// TIA Portal project "progetto KENNEDY_ok" (V16)

(* hardware
DEVICE "HMI_1"  KTP900 Basic PN
   slot 0: "HMI_1"  KTP900 Basic PN  6AV2 123-2JB03-0AX0  15.1.0.0
   slot 1: "HMI_RT_1"  KTP900 Basic PN  6AV2 123-2JB03-0AX0  15.1.0.0
   slot 5: "HMI_1.IE_CP_1"  PROFINET Interface  15.0.1.0
      slot 1: "Interfaccia_1 PROFINET"  PROFINET Interface
         slot 1: "Porta_1"  Port
DEVICE "S7-1200 station_1"  S7-1200 Station
   slot 0: "Telaio di montaggio_0"  S7-1200 Rack  Rack  V1.0
   slot 1: "PLC_1"  CPU 1212C DC/DC/DC  6ES7 212-1AE40-0XB0  V4.4
*)

// ===== PLC "PLC_1"  CPU 1212C DC/DC/DC =====

VAR_GLOBAL   // PLC tag table "Tabella delle variabili standard"
   "EV PISTONE 1 MISURA" AT %Q0.2 : Bool;
   "EV PINZA" AT %Q0.5 : Bool;
   "EV PISTONE 3 SU GIU" AT %Q0.4 : Bool;
   "EV PISTONE 2 MISURA" AT %Q0.3 : Bool;
   "EV AV INDIETRO RIEMPITRICE" AT %Q0.6 : Bool;
   "EV BECCUCCIO RIEMPITRICE" AT %Q0.7 : Bool;
   "EV RIEMPIMENTO FLACONE" AT %Q8.0 : Bool;
   "RISERVA 2" AT %I0.7 : Bool;
   "FC PISTONE 1 AVANTI" AT %I8.3 : Bool;
   "FC PISTONE 1 INDIETRO" AT %I8.4 : Bool;
   "FC PISTONE 2 AVANTI" AT %I8.5 : Bool;
   "FC PISTONE 2 INDIETRO" AT %I8.6 : Bool;
   "FC PISTONE 3 VERTICALE GIU" AT %I8.7 : Bool;
   "FC PISTONE 3 VERTICALE SU" AT %I9.0 : Bool;
   "FC PISTONE 4 PINZA APERTA" AT %I9.1 : Bool;
   "FC SENSORE PRESENZA PEZZO AL CARICO" AT %I9.2 : Bool;
   "FUNGO EMERGENZA" AT %I0.0 : Bool;
   "PULSANTE RESET EMERGENZA" AT %I0.1 : Bool;
   "SELETTORE MANU  AUTO" AT %I0.3 : Bool;
   "PULSANTE START CICLO" AT %I0.4 : Bool;
   "PULSANTE STOP CICLO" AT %I0.5 : Bool;
   "RISERVA 1" AT %I0.6 : Bool;
   "PULSANTE 1" AT %I8.0 : Bool;
   "PULSANTE 2" AT %I8.1 : Bool;
   "LAMPADA RESET EMERGENZA" AT %Q0.0 : Bool;
   "LAMPADA PULSANTE START VERDE" AT %Q0.1 : Bool;
   "SELETTORE 1" AT %I0.2 : Bool;
   "FC AVANTI RIEMPITRICE" AT %I9.4 : Bool;
   "RISERVA 3" AT %I8.2 : Bool;
   "FC INDIETRO RIEMPITRICE" AT %I9.5 : Bool;
   "FC GIU BECCUCCIO RIEMPITRICE" AT %I9.6 : Bool;
   "FC SU BECCUCCIO RIEMPITRICE" AT %I9.7 : Bool;
   "Clock_Byte" AT %MB0 : Byte;
   "Clock_10Hz" AT %M0.0 : Bool;
   "Clock_5Hz" AT %M0.1 : Bool;
   "Clock_2.5Hz" AT %M0.2 : Bool;
   "Clock_2Hz" AT %M0.3 : Bool;
   "Clock_1.25Hz" AT %M0.4 : Bool;
   "Clock_1Hz" AT %M0.5 : Bool;
   "Clock_0.625Hz" AT %M0.6 : Bool;
   "Clock_0.5Hz" AT %M0.7 : Bool;
   "RISERVA 4" AT %I9.3 : Bool;
END_VAR

DATA_BLOCK "0-DB-Generale"   // DB4
{ S7_Optimized_Access := 'TRUE' }
VERSION : 0.1
   VAR
      "0-COMMENTO" : Bool;   // Usata per decommentare righe di ladder
      "0-TEST" : Bool;   // Usata per simulare una uscita finta nei test
      "0-IdCommessa" : Int;   // Identificiativo della commessa (ipoteticamente) ricevuta dal pc bordo macchina
      "0-IdMacchinario" : Int;   // Int da fissare costante all'interno della macchina. Identifica univocamente il PLC, ma noi ne abbiamo uno solo
      "0-IdProdotto" : Int;   // Identificativo del prodotto (ipoteticamente) commissionato dall'ufficio
      "0-PezziTotali" : Int;   // Il numero toale di pezzi da produrre (ipoteticamente impostato da ufficio)
      "0-TimeStampAttuale" : DTL;   // Il tempo reale del plc
      "0-PezziBuoniProdotti" : Int;   // Il numero di pezzi non difettati prodotti
      "0-PezziScartiProdotti" : Int;   // Il numero di pezzi fallati prodotti
      "0-StatoMacchina" : Int;   // L'intero in sostituziona all'enum che identifica lo stato macchina: viene gestito (prelevato tramite OPC Ua e scritto in SQL Server) nel codice c#. Legenda: 0 - Verde, Stato Start; 1 - Rosso, Stato Fermo; 2 - Giallo, Stato Pronto;
      "0-MinutiDiLavoro" : Int;   // I minuti totali di lavoro del macchinario: sono dati dall'accumulo delle differenze tra TImeStampFineCiclo e TImeStampInizioCiclo alla fine di ogni ciclo
      "0-TImeStampInizioCiclo" : Int;   // TimeStamp al momento dell'inizio del ciclo di una data commessa
      "0-TimeStampFineCiclo" : Int;   // TimeStamp al momento della fine del ciclo di una data commessa
      "0-IdAttuatori" : Array[0..1] of Int;   // Id univoco per ciascun pistoni in questo PLC (idealmente potrebbe tracciare anche singole parti meccaniche come viti ecc. ecc.). E' analogo al mac address delle schede di rete nei pc per intendersi.
      "0-NumeroAttivazioniAttuatori" : Array[0..1] of Int;   // Array che contiene l'accumulatore delle attivazioni degli attuatori per ciascun attuatore. In altre parole mi immagino una matrice con una riga con l'array degli attuatori e una riga sotto con l'accumulo delle attivazioni per ogni attuatore
      "0-IdSensori" : Array[0..1] of Int;   // Analogo agli attuatori: vedi loro commenti
      "0-NumeroAttivazioniSensori" : Array[0..1] of Int;   // Analogo agli attuatori: vedi loro commenti
      "0-PezziPerMinuto" : Real;   // Usiamo l'equivalente PLC del float. Per standard contrattuali e' buona pratica usare il tipo REAL per le velocita' al minuto
      "0-Allarmi" : Array[0..1] of Bool;   // Attivazione o Meno di ogni allarme (logica simile alla matrice deglia attuatori: vedi commenti sopra)
      "1-NonEmergenza" : Bool;   // NonEmergenza = True = macchina in regolare funzione, NonEmergenza = False = macchina in emergenza e ferma
      "3-AvvioCicloAuto" : Bool;   // Il ciclo automatico si avvia
      "3-CicloAutoPronto" : Bool;   // Il ciclo automatico e' pronto per l'avvio
      "3-MacchinaInPosizioneDiPartenza" : Bool;   // Risultato logico combinatorio sui finecorsa (se sono tutti nelle opportune posizioni la macchina e' nella posizione iniziale)
      "3-GestioneManuPronta" : Bool;   // La gestione manuale dell'automazione da hmi e' pronta per essere usata
      "3-AvvioGestioneManu" : Bool;   // La gestione manuale si avvia
      "4-ResetMacchinaInPosizioneDiPartenza" : Bool;   // Resetta le posizioni dei pistoni alla fine del ciclo
      "4-Passo1" : Bool;   // Il pistone 3 si abbassa sul flacone (pre riempimento)
      "4-Passo2" : Bool;   // Il pistone Pinza si chiude sul flacone (pre riempimento)
      "4-Passo3" : Bool;   // Il pistone 3 si alza con il flacone (pre riempimento)
      "4-Passo4" : Bool;   // Il pistone 2 si estende a destra (pre riempimento)
      "4-Passo5" : Bool;   // Il pistone 1 si estende a destra (pre riempimento)
      "4-Passo6" : Bool;   // Il pistone 3 si abbassa con il flacone (pre riempimento)
      "4-Passo7" : Bool;   // Il pistone pinza si apre con il flacone (pre riempimento)
      "4-Passo8" : Bool;   // Il pistone 3 si alza senza flacone in attesa del riempimento (pre riempimento)
      "4-Passo9" : Bool;   // Il pistone riempitore 1 si estende a sinistra
      "4-Passo10" : Bool;   // Il pistone riempitore 2 abbassa il beccuccio
      "4-Passo11" : Bool;   // Il pistone riempitore 2 alza il beccuccio
      "4-Passo12" : Bool;   // Il pistone riempitore 1 rientra a destra
      "4-Passo13" : Bool;   // Il pistone 3 scende sopra al flacone (post riempimento)
      "4-Passo14" : Bool;   // Il pistone Pinza si chiude sul flacone (post riempimento)
      "4-Passo15" : Bool;   // Il pistone 3 si alza con il flacone (post riempimento)
      "4-Passo16" : Bool;   // Il pistone 2 si ritrae con il flacone (post riempimento)
      "4-Passo17" : Bool;   // Il pistone 3 si abbassa sulla zona di scarico
      "4-Passo18" : Bool;   // Il pistone Pinza si apre
      "4-Passo19" : Bool;   // Il pistone 3 si alza dalla zona di scarico
      "4-Passo20" : Bool;   // Il pistone 1 si ritrae nella posizione di partenza: il ciclo è finito
      "5-HMI => Only current time" : Time_Of_Day;   // Ora corrente (time) estrapolata dal dato totale (Time of Day)
      "5-HMI => Only current date" : Date;   // Data corrente (date) estrapolata dal dato totale (Time of Day)
      "5-HMI => Current time of day" : DTL;   // Current Time of Day include tutti i dati temporali all'acquisizione, è una sorta di TimeStamp, tipo dato DTL
      "5-HMI => Timer ultima eccezione" : Bool;   // Variabile che gestisce l'obbligo di esecuzione del login: compare un messaggio temporizzato a 5s ogni volta che si cliccano elementi cliccabili nell'HMI senza effettuare il login
      "5-ErroriDiConversione" : Int;   // Qui vengono ritornati gli interi che indicano eventuali errori nella conversione ed estrazione di data o ora dalla DTL che contiene tutto il timestamp. Se la conversione avviene con successo il valore di questa variabile è 0000
      "5-VisibilitaComandiManuali" : Bool;   // Gestisce la visibilita' dell'automazione per la schermata manuale dell'hmi. In base allo stato della variabile si vede il manipolatore o la riempitrice.
      "6-Pistone-1-Manuale" : Bool;   // Variabile d'appoggio a sostituire l'uscita diretta nel blocco ciclo manuale
      "6-Pistone-2-Manuale" : Bool;   // Variabile d'appoggio a sostituire l'uscita diretta nel blocco ciclo manuale
      "6-Pistone-3-Manuale" : Bool;   // Variabile d'appoggio a sostituire l'uscita diretta nel blocco ciclo manuale
      "6-Pistone-4-(Pinza)-Manuale" : Bool;   // Variabile d'appoggio a sostituire l'uscita diretta nel blocco ciclo manuale
      "6-Pistone-5-(Riempitrice)-Manuale" : Bool;   // Variabile d'appoggio a sostituire l'uscita diretta nel blocco ciclo manuale
      "6-Beccuccio-(Riempitrice)-Manuale" : Bool;   // Variabile d'appoggio a sostituire l'uscita diretta nel blocco ciclo manuale
      "6-Riempimento-(Riempitrice)-Manuale" : Bool;   // Variabile d'appoggio a sostituire l'uscita diretta nel blocco ciclo manuale
      "6-PulsanteAvantiPistone1" : Bool;   // Variabile d'appoggio che identifica il relativo tasto dell'HMI nel blocco uscite
      "6-PulsanteIndietroPistone1" : Bool;   // Variabile d'appoggio che identifica il relativo tasto dell'HMI nel blocco uscite
      "6-PulsanteAvantiPistone2" : Bool;   // Variabile d'appoggio che identifica il relativo tasto dell'HMI nel blocco uscite
      "6-PulsanteIndietroPistone2" : Bool;   // Variabile d'appoggio che identifica il relativo tasto dell'HMI nel blocco uscite
      "6-PulsanteGiuPistone3" : Bool;   // Variabile d'appoggio che identifica il relativo tasto dell'HMI nel blocco uscite
      "6-PulsanteSuPistone3" : Bool;   // Variabile d'appoggio che identifica il relativo tasto dell'HMI nel blocco uscite
      "6-PulsanteChiudiPinza" : Bool;   // Variabile d'appoggio che identifica il relativo tasto dell'HMI nel blocco uscite
      "6-PulsanteApriPinza" : Bool;   // Variabile d'appoggio che identifica il relativo tasto dell'HMI nel blocco uscite
      "6-PulsanteAvantiPistone5Riempitrice" : Bool;   // Variabile d'appoggio che identifica il relativo tasto dell'HMI nel blocco uscite
      "6-PulsanteIndietroPistone5Riempitrice" : Bool;   // Variabile d'appoggio che identifica il relativo tasto dell'HMI nel blocco uscite
      "6-PulsanteGiuPistone6Beccuccio" : Bool;   // Variabile d'appoggio che identifica il relativo tasto dell'HMI nel blocco uscite
      "6-PulsanteSuPistone6Beccuccio" : Bool;   // Variabile d'appoggio che identifica il relativo tasto dell'HMI nel blocco uscite
      "6-PulsanteRiempimento" : Bool;
   END_VAR
BEGIN
END_DATA_BLOCK

// folder: RISERVATO_NON_MODIFICARE

DATA_BLOCK "Blocco_dati_1"   // DB1
{ S7_Optimized_Access := 'TRUE' }
VERSION : 0.1
   VAR
      "pistone 1  X" : Int;
      "pistone 1  Y" : Int;
      "pistone 2  X" : Int;
      "pistone 2 Y" : Int;
      "stelo pistone 2 x" : Int;
      "stelo pistone 2 y" : Int;
      "pistone 3  X" : Int;
      "pistone 3 Y" : Int;
      "stelo pistone 3 x" : Int;
      "stelo pistone 3 y" : Int;
      "corpo pinza x" : Int;
      "corpo pinza y" : Int;
      "dita aperte x" : Int;
      "dita aperte y" : Int;
      "dita chiuse x" : Int;
      "dita chiuse y" : Int;
      "pistone riempitore av ind x" : Int;
      "pistone riempitore av ind y" : Int;
      "riempitore av ind x" : Int;
      "riempitore su giu y" : Int;
      "flacone x" : Int;
      "flacone y" : Int;
      "riempimento flacone" : Int;
      "pinza aperta" : Int;
      "pinza chiusa" : Int;
      "fungo emergenza" : Bool;
      "reset emergenza" : Bool;
      "lampada emergenza" : Bool;
      "pulsante start ciclo" : Bool;
      "lampada pulsante start ciclo" : Bool;
      "selettore 1 leva corta" : Bool;
      "selettore auto manu" : Bool;
      "pulsante 1" : Bool;
      "pulsante 2" : Bool;
      "pulsante stop ciclo" : Bool;
      MANUALI : Byte;
      "FLACONE PIENO" : Bool;
      "FLACONE PRESO" : Bool;
      "FLACONE IN RIEMPIMENTO" : Bool;
      "SENSORE SU" : Byte;
      "SENSORE GIU" : Byte;
      "SENSORE PINZA APERTA" : Byte;
      "SENSORE INDIETRO PISTONE_1" : Byte;
      "SENSORE AVANTI PISTONE_1" : Byte;
      "SENSORE INDIETRO PISTONE_2" : Byte;
      "SENSORE AVANTI PISTONE_2" : Byte;
      "SENSORE INDIETRO PISTONE_3" : Byte;
      "SENSORE AVANTI PISTONE_3" : Byte;
      "SENSORE INDIETRO RIEMPITRICE" : Byte;
      "SENSORE AVANTI RIEMPITRICE" : Byte;
      "SENSORE SU RIEMPITRICE" : Byte;
      "SENSORE GIU RIEMPITRICE" : Byte;
      "SENSORE PRESENZA FLACONE" : Bool;
      "RISPOSTA TELECAMERA DI ISPEZIONE" : Byte;
      "APPOGGIO PARTENZA" : Bool;
      "SELETTORE SIMULAZIONE PRESENZA PEZZO AL CARICO" : Bool;
      "VISUALIZZA IL FLACONE" : Bool;
   END_VAR
BEGIN
END_DATA_BLOCK

// folder: System blocks/Program resources

DATA_BLOCK "IEC_Timer_0_DB"   // DB2
{ S7_Optimized_Access := 'TRUE' }
AUTHOR : Simatic
FAMILY : IEC
NAME : IEC_TMR
VERSION : 1.0
// stored: InstanceOfName IEC_TIMER
"IEC_TIMER"
BEGIN
END_DATA_BLOCK

DATA_BLOCK "azzerooo"   // DB3
{ S7_Optimized_Access := 'TRUE' }
AUTHOR : Simatic
FAMILY : IEC
NAME : IEC_TMR
VERSION : 1.0
// stored: InstanceOfName IEC_TIMER
"IEC_TIMER"
BEGIN
END_DATA_BLOCK

DATA_BLOCK "IEC_Timer_0_DB_3"   // DB5
{ S7_Optimized_Access := 'TRUE' }
AUTHOR : Simatic
FAMILY : IEC
NAME : IEC_TMR
VERSION : 1.0
// stored: InstanceOfName IEC_TIMER
"IEC_TIMER"
BEGIN
END_DATA_BLOCK

DATA_BLOCK "IEC_Timer_0_DB_4"   // DB6
{ S7_Optimized_Access := 'TRUE' }
AUTHOR : Simatic
FAMILY : IEC
NAME : IEC_TMR
VERSION : 1.0
// stored: InstanceOfName IEC_TIMER
"IEC_TIMER"
BEGIN
END_DATA_BLOCK

DATA_BLOCK "IEC_Timer_0_DB_5"   // DB7
{ S7_Optimized_Access := 'TRUE' }
AUTHOR : Simatic
FAMILY : IEC
NAME : IEC_TMR
VERSION : 1.0
// stored: InstanceOfName IEC_TIMER
"IEC_TIMER"
BEGIN
END_DATA_BLOCK

DATA_BLOCK "IEC_Timer_0_DB_6"   // DB8
{ S7_Optimized_Access := 'TRUE' }
AUTHOR : Simatic
FAMILY : IEC
NAME : IEC_TMR
VERSION : 1.0
// stored: InstanceOfName IEC_TIMER
"IEC_TIMER"
BEGIN
END_DATA_BLOCK

DATA_BLOCK "IEC_Timer_0_DB_7"   // DB9
{ S7_Optimized_Access := 'TRUE' }
AUTHOR : Simatic
FAMILY : IEC
NAME : IEC_TMR
VERSION : 1.0
// stored: InstanceOfName IEC_TIMER
"IEC_TIMER"
BEGIN
END_DATA_BLOCK

DATA_BLOCK "IEC_Timer_0_DB_8"   // DB10
{ S7_Optimized_Access := 'TRUE' }
AUTHOR : Simatic
FAMILY : IEC
NAME : IEC_TMR
VERSION : 1.0
// stored: InstanceOfName IEC_TIMER
"IEC_TIMER"
BEGIN
END_DATA_BLOCK

DATA_BLOCK "IEC_Timer_0_DB_9"   // DB11
{ S7_Optimized_Access := 'TRUE' }
AUTHOR : Simatic
FAMILY : IEC
NAME : IEC_TMR
VERSION : 1.0
// stored: InstanceOfName IEC_TIMER
"IEC_TIMER"
BEGIN
END_DATA_BLOCK

DATA_BLOCK "IEC_Timer_0_DB_10"   // DB12
{ S7_Optimized_Access := 'TRUE' }
AUTHOR : Simatic
FAMILY : IEC
NAME : IEC_TMR
VERSION : 1.0
// stored: InstanceOfName IEC_TIMER
"IEC_TIMER"
BEGIN
END_DATA_BLOCK

DATA_BLOCK "IEC_Timer_0_DB_11"   // DB13
{ S7_Optimized_Access := 'TRUE' }
AUTHOR : Simatic
FAMILY : IEC
NAME : IEC_TMR
VERSION : 1.0
// stored: InstanceOfName IEC_TIMER
"IEC_TIMER"
BEGIN
END_DATA_BLOCK

DATA_BLOCK "IEC_Timer_0_DB_12"   // DB14
{ S7_Optimized_Access := 'TRUE' }
AUTHOR : Simatic
FAMILY : IEC
NAME : IEC_TMR
VERSION : 1.0
// stored: InstanceOfName IEC_TIMER
"IEC_TIMER"
BEGIN
END_DATA_BLOCK

DATA_BLOCK "IEC_Timer_0_DB_13"   // DB15
{ S7_Optimized_Access := 'TRUE' }
AUTHOR : Simatic
FAMILY : IEC
NAME : IEC_TMR
VERSION : 1.0
// stored: InstanceOfName IEC_TIMER
"IEC_TIMER"
BEGIN
END_DATA_BLOCK

DATA_BLOCK "IEC_Timer_0_DB_1"   // DB16
{ S7_Optimized_Access := 'TRUE' }
AUTHOR : Simatic
FAMILY : IEC
NAME : IEC_TMR
VERSION : 1.0
// stored: InstanceOfName IEC_TIMER
"IEC_TIMER"
BEGIN
END_DATA_BLOCK

DATA_BLOCK "IEC_Timer_0_DB_2"   // DB17
{ S7_Optimized_Access := 'TRUE' }
AUTHOR : Simatic
FAMILY : IEC
NAME : IEC_TMR
VERSION : 1.0
// stored: InstanceOfName IEC_TIMER
"IEC_TIMER"
BEGIN
END_DATA_BLOCK

DATA_BLOCK "IEC_Timer_0_DB_14"   // DB18
{ S7_Optimized_Access := 'TRUE' }
AUTHOR : Simatic
FAMILY : IEC
NAME : IEC_TMR
VERSION : 1.0
// stored: InstanceOfName IEC_TIMER
"IEC_TIMER"
BEGIN
END_DATA_BLOCK

DATA_BLOCK "IEC_Timer_0_DB_15"   // DB19
{ S7_Optimized_Access := 'TRUE' }
AUTHOR : Simatic
FAMILY : IEC
NAME : IEC_TMR
VERSION : 1.0
// stored: InstanceOfName IEC_TIMER
"IEC_TIMER"
BEGIN
END_DATA_BLOCK

DATA_BLOCK "IEC_Timer_0_DB_16"   // DB20
{ S7_Optimized_Access := 'TRUE' }
AUTHOR : Simatic
FAMILY : IEC
NAME : IEC_TMR
VERSION : 1.0
// stored: InstanceOfName IEC_TIMER
"IEC_TIMER"
BEGIN
END_DATA_BLOCK

DATA_BLOCK "IEC_Timer_0_DB_17"   // DB21
{ S7_Optimized_Access := 'TRUE' }
AUTHOR : Simatic
FAMILY : IEC
NAME : IEC_TMR
VERSION : 1.0
// stored: InstanceOfName IEC_TIMER
"IEC_TIMER"
BEGIN
END_DATA_BLOCK

DATA_BLOCK "IEC_Timer_0_DB_18"   // DB22
{ S7_Optimized_Access := 'TRUE' }
AUTHOR : Simatic
FAMILY : IEC
NAME : IEC_TMR
VERSION : 1.0
// stored: InstanceOfName IEC_TIMER
"IEC_TIMER"
BEGIN
END_DATA_BLOCK

DATA_BLOCK "IEC_Timer_0_DB_19"   // DB23
{ S7_Optimized_Access := 'TRUE' }
AUTHOR : Simatic
FAMILY : IEC
NAME : IEC_TMR
VERSION : 1.0
// stored: InstanceOfName IEC_TIMER
"IEC_TIMER"
BEGIN
END_DATA_BLOCK

DATA_BLOCK "IEC_Timer_0_DB_20"   // DB24
{ S7_Optimized_Access := 'TRUE' }
AUTHOR : Simatic
FAMILY : IEC
NAME : IEC_TMR
VERSION : 1.0
// stored: InstanceOfName IEC_TIMER
"IEC_TIMER"
BEGIN
END_DATA_BLOCK

DATA_BLOCK "IEC_Timer_0_DB_21"   // DB25
{ S7_Optimized_Access := 'TRUE' }
AUTHOR : Simatic
FAMILY : IEC
NAME : IEC_TMR
VERSION : 1.0
// stored: InstanceOfName IEC_TIMER
"IEC_TIMER"
BEGIN
END_DATA_BLOCK

DATA_BLOCK "IEC_Timer_0_DB_22"   // DB26
{ S7_Optimized_Access := 'TRUE' }
AUTHOR : Simatic
FAMILY : IEC
NAME : IEC_TMR
VERSION : 1.0
// stored: InstanceOfName IEC_TIMER
"IEC_TIMER"
BEGIN
END_DATA_BLOCK

DATA_BLOCK "IEC_Timer_0_DB_23"   // DB27
{ S7_Optimized_Access := 'TRUE' }
AUTHOR : Simatic
FAMILY : IEC
NAME : IEC_TMR
VERSION : 1.0
// stored: InstanceOfName IEC_TIMER
"IEC_TIMER"
BEGIN
END_DATA_BLOCK

DATA_BLOCK "IEC_Timer_0_DB_24"   // DB28
{ S7_Optimized_Access := 'TRUE' }
AUTHOR : Simatic
FAMILY : IEC
NAME : IEC_TMR
VERSION : 1.0
// stored: InstanceOfName IEC_TIMER
"IEC_TIMER"
BEGIN
END_DATA_BLOCK

DATA_BLOCK "IEC_Timer_0_DB_25"   // DB29
{ S7_Optimized_Access := 'TRUE' }
AUTHOR : Simatic
FAMILY : IEC
NAME : IEC_TMR
VERSION : 1.0
// stored: InstanceOfName IEC_TIMER
"IEC_TIMER"
BEGIN
END_DATA_BLOCK

DATA_BLOCK "IEC_Timer_0_DB_26"   // DB30
{ S7_Optimized_Access := 'TRUE' }
AUTHOR : Simatic
FAMILY : IEC
NAME : IEC_TMR
VERSION : 1.0
// stored: InstanceOfName IEC_TIMER
"IEC_TIMER"
BEGIN
END_DATA_BLOCK

DATA_BLOCK "IEC_Timer_0_DB_27"   // DB31
{ S7_Optimized_Access := 'TRUE' }
AUTHOR : Simatic
FAMILY : IEC
NAME : IEC_TMR
VERSION : 1.0
// stored: InstanceOfName IEC_TIMER
"IEC_TIMER"
BEGIN
END_DATA_BLOCK

DATA_BLOCK "IEC_Timer_0_DB_28"   // DB32
{ S7_Optimized_Access := 'TRUE' }
AUTHOR : Simatic
FAMILY : IEC
NAME : IEC_TMR
VERSION : 1.0
// stored: InstanceOfName IEC_TIMER
"IEC_TIMER"
BEGIN
END_DATA_BLOCK

DATA_BLOCK "IEC_Timer_0_DB_29"   // DB33
{ S7_Optimized_Access := 'TRUE' }
AUTHOR : Simatic
FAMILY : IEC
NAME : IEC_TMR
VERSION : 1.0
// stored: InstanceOfName IEC_TIMER
"IEC_TIMER"
BEGIN
END_DATA_BLOCK

DATA_BLOCK "IEC_Timer_0_DB_30"   // DB34
{ S7_Optimized_Access := 'TRUE' }
AUTHOR : Simatic
FAMILY : IEC
NAME : IEC_TMR
VERSION : 1.0
// stored: InstanceOfName IEC_TIMER
"IEC_TIMER"
BEGIN
END_DATA_BLOCK

DATA_BLOCK "IEC_Timer_0_DB_31"   // DB35
{ S7_Optimized_Access := 'TRUE' }
AUTHOR : Simatic
FAMILY : IEC
NAME : IEC_TMR
VERSION : 1.0
// stored: InstanceOfName IEC_TIMER
"IEC_TIMER"
BEGIN
END_DATA_BLOCK

DATA_BLOCK "IEC_Timer_0_DB_32"   // DB36
{ S7_Optimized_Access := 'TRUE' }
AUTHOR : Simatic
FAMILY : IEC
NAME : IEC_TMR
VERSION : 1.0
// stored: InstanceOfName IEC_TIMER
"IEC_TIMER"
BEGIN
END_DATA_BLOCK

DATA_BLOCK "IEC_Timer_0_DB_33"   // DB37
{ S7_Optimized_Access := 'TRUE' }
AUTHOR : Simatic
FAMILY : IEC
NAME : IEC_TMR
VERSION : 1.0
// stored: InstanceOfName IEC_TIMER
"IEC_TIMER"
BEGIN
END_DATA_BLOCK

DATA_BLOCK "IEC_Timer_0_DB_34"   // DB38
{ S7_Optimized_Access := 'TRUE' }
AUTHOR : Simatic
FAMILY : IEC
NAME : IEC_TMR
VERSION : 1.0
// stored: InstanceOfName IEC_TIMER
"IEC_TIMER"
BEGIN
END_DATA_BLOCK

// folder: (top level)

FUNCTION "1-Allarmi" : Void   // FC2, LAD
{ S7_Optimized_Access := 'TRUE' }
VERSION : 0.1
BEGIN

REGION Network 1: NonEmergenza = True = macchina in regolare funzione, NonEmergenza = False = macchina in emergenza e ferma
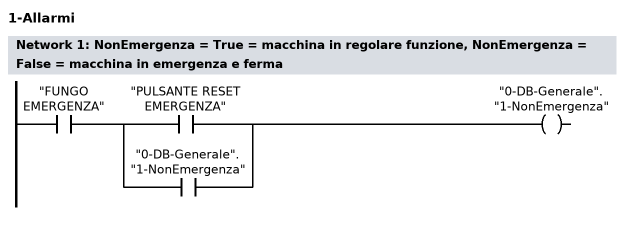
   RUNG wire#powerrail
      Contact( "FUNGO EMERGENZA" )
      wire#w1
      Contact( "PULSANTE RESET EMERGENZA" )
      wire#w2
      Coil( "0-DB-Generale"."1-NonEmergenza" )
   END_RUNG
   RUNG wire#w1
      Contact( "0-DB-Generale"."1-NonEmergenza" )
   END_RUNG wire#w2
   // the same network as SCL:
   "0-DB-Generale"."1-NonEmergenza" := "FUNGO EMERGENZA" AND ("PULSANTE RESET EMERGENZA" OR "0-DB-Generale"."1-NonEmergenza");
END_REGION
END_FUNCTION

FUNCTION "2-Uscite" : Void   // FC3, LAD
{ S7_Optimized_Access := 'TRUE' }
VERSION : 0.1
BEGIN

REGION Network 1: USCITA %Q0.0 - LAMPADA DI EMERGENZA
   // Descr: 
   // Who: Gestione prima uscita cablata.
   // What: Se la macchina non è in emergenza la lampada non si accende e viceversa.
   // How: Verifica mediante test ladder True If Off (--|/|--, NC) sulla variabile booleana (bit) associata allo stato di emergenza. Se il fungo viene usato lo stato di NonEmergenza passa da 1 a 0, da true a false quindi qui il True If Off lascia passare il segnale attivando la lampada reset di emergenza.
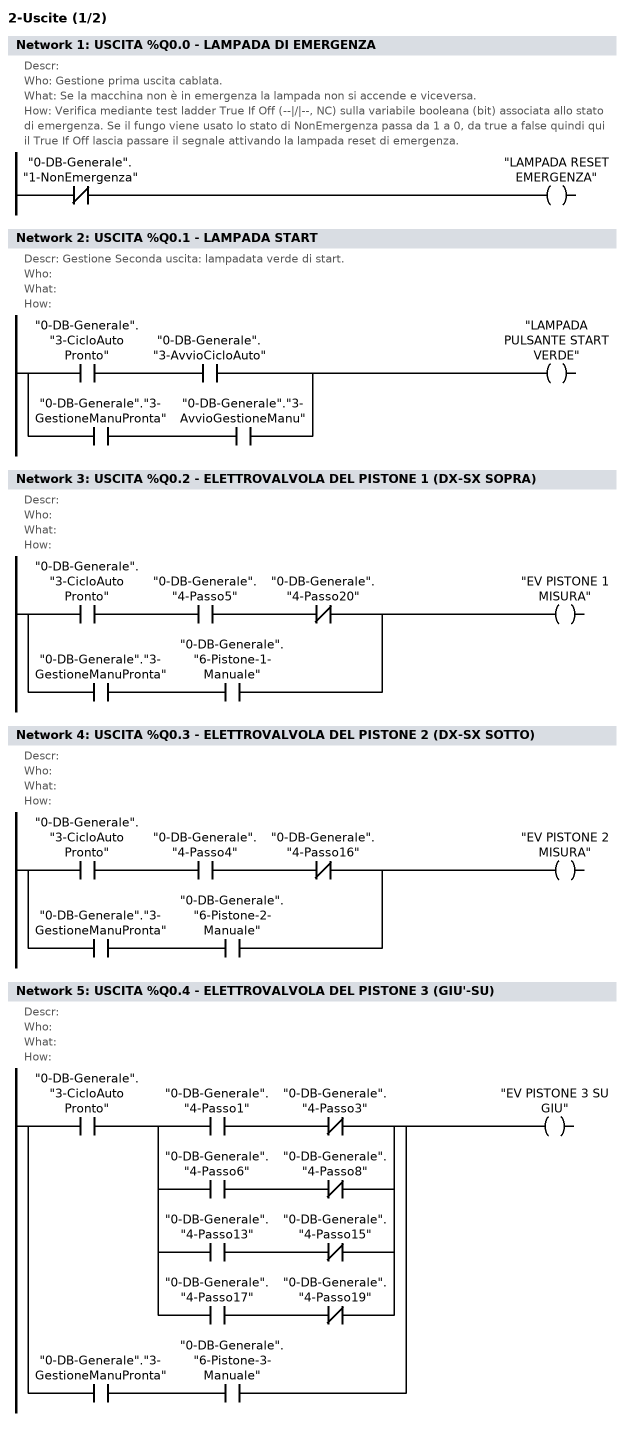
   RUNG wire#powerrail
      I_Contact( "0-DB-Generale"."1-NonEmergenza" )
      Coil( "LAMPADA RESET EMERGENZA" )
   END_RUNG
   // the same network as SCL:
   "LAMPADA RESET EMERGENZA" := NOT "0-DB-Generale"."1-NonEmergenza";
END_REGION

REGION Network 2: USCITA %Q0.1 - LAMPADA START
   // Descr: Gestione Seconda uscita: lampadata verde di start.
   // Who: 
   // What: 
   // How:
   RUNG wire#powerrail
      Contact( "0-DB-Generale"."3-CicloAutoPronto" )
      Contact( "0-DB-Generale"."3-AvvioCicloAuto" )
      wire#w1
      Coil( "LAMPADA PULSANTE START VERDE" )
   END_RUNG
   RUNG wire#powerrail
      Contact( "0-DB-Generale"."3-GestioneManuPronta" )
      Contact( "0-DB-Generale"."3-AvvioGestioneManu" )
   END_RUNG wire#w1
   // the same network as SCL:
   "LAMPADA PULSANTE START VERDE" := ("0-DB-Generale"."3-CicloAutoPronto" AND "0-DB-Generale"."3-AvvioCicloAuto") OR ("0-DB-Generale"."3-GestioneManuPronta" AND "0-DB-Generale"."3-AvvioGestioneManu");
END_REGION

REGION Network 3: USCITA %Q0.2 - ELETTROVALVOLA DEL PISTONE 1 (DX-SX SOPRA)
   // Descr: 
   // Who: 
   // What: 
   // How:
   RUNG wire#powerrail
      Contact( "0-DB-Generale"."3-CicloAutoPronto" )
      Contact( "0-DB-Generale"."4-Passo5" )
      I_Contact( "0-DB-Generale"."4-Passo20" )
      wire#w1
      Coil( "EV PISTONE 1 MISURA" )
   END_RUNG
   RUNG wire#powerrail
      Contact( "0-DB-Generale"."3-GestioneManuPronta" )
      Contact( "0-DB-Generale"."6-Pistone-1-Manuale" )
   END_RUNG wire#w1
   // the same network as SCL:
   "EV PISTONE 1 MISURA" := ("0-DB-Generale"."3-CicloAutoPronto" AND "0-DB-Generale"."4-Passo5" AND NOT "0-DB-Generale"."4-Passo20") OR ("0-DB-Generale"."3-GestioneManuPronta" AND "0-DB-Generale"."6-Pistone-1-Manuale");
END_REGION

REGION Network 4: USCITA %Q0.3 - ELETTROVALVOLA DEL PISTONE 2 (DX-SX SOTTO)
   // Descr: 
   // Who: 
   // What: 
   // How:
   RUNG wire#powerrail
      Contact( "0-DB-Generale"."3-CicloAutoPronto" )
      Contact( "0-DB-Generale"."4-Passo4" )
      I_Contact( "0-DB-Generale"."4-Passo16" )
      wire#w1
      Coil( "EV PISTONE 2 MISURA" )
   END_RUNG
   RUNG wire#powerrail
      Contact( "0-DB-Generale"."3-GestioneManuPronta" )
      Contact( "0-DB-Generale"."6-Pistone-2-Manuale" )
   END_RUNG wire#w1
   // the same network as SCL:
   "EV PISTONE 2 MISURA" := ("0-DB-Generale"."3-CicloAutoPronto" AND "0-DB-Generale"."4-Passo4" AND NOT "0-DB-Generale"."4-Passo16") OR ("0-DB-Generale"."3-GestioneManuPronta" AND "0-DB-Generale"."6-Pistone-2-Manuale");
END_REGION

REGION Network 5: USCITA %Q0.4 - ELETTROVALVOLA DEL PISTONE 3 (GIU'-SU)
   // Descr: 
   // Who: 
   // What: 
   // How:
   RUNG wire#powerrail
      Contact( "0-DB-Generale"."3-CicloAutoPronto" )
      wire#w1
      Contact( "0-DB-Generale"."4-Passo1" )
      I_Contact( "0-DB-Generale"."4-Passo3" )
      wire#w2
      Coil( "EV PISTONE 3 SU GIU" )
   END_RUNG
   RUNG wire#w1
      Contact( "0-DB-Generale"."4-Passo6" )
      I_Contact( "0-DB-Generale"."4-Passo8" )
   END_RUNG wire#w2
   RUNG wire#w1
      Contact( "0-DB-Generale"."4-Passo13" )
      I_Contact( "0-DB-Generale"."4-Passo15" )
   END_RUNG wire#w2
   RUNG wire#w1
      Contact( "0-DB-Generale"."4-Passo17" )
      I_Contact( "0-DB-Generale"."4-Passo19" )
   END_RUNG wire#w2
   RUNG wire#powerrail
      Contact( "0-DB-Generale"."3-GestioneManuPronta" )
      Contact( "0-DB-Generale"."6-Pistone-3-Manuale" )
   END_RUNG wire#w2
   // the same network as SCL:
   "EV PISTONE 3 SU GIU" := ("0-DB-Generale"."3-CicloAutoPronto" AND (("0-DB-Generale"."4-Passo1" AND NOT "0-DB-Generale"."4-Passo3") OR ("0-DB-Generale"."4-Passo6" AND NOT "0-DB-Generale"."4-Passo8") OR ("0-DB-Generale"."4-Passo13" AND NOT "0-DB-Generale"."4-Passo15") OR ("0-DB-Generale"."4-Passo17" AND NOT "0-DB-Generale"."4-Passo19"))) OR ("0-DB-Generale"."3-GestioneManuPronta" AND "0-DB-Generale"."6-Pistone-3-Manuale");
END_REGION

REGION Network 6: USCITA %Q0.5 - ELETTROVALVOLA DELLA PINZA (APRI-CHIUDI)
   // Descr: 
   // Who: 
   // What: 
   // How:
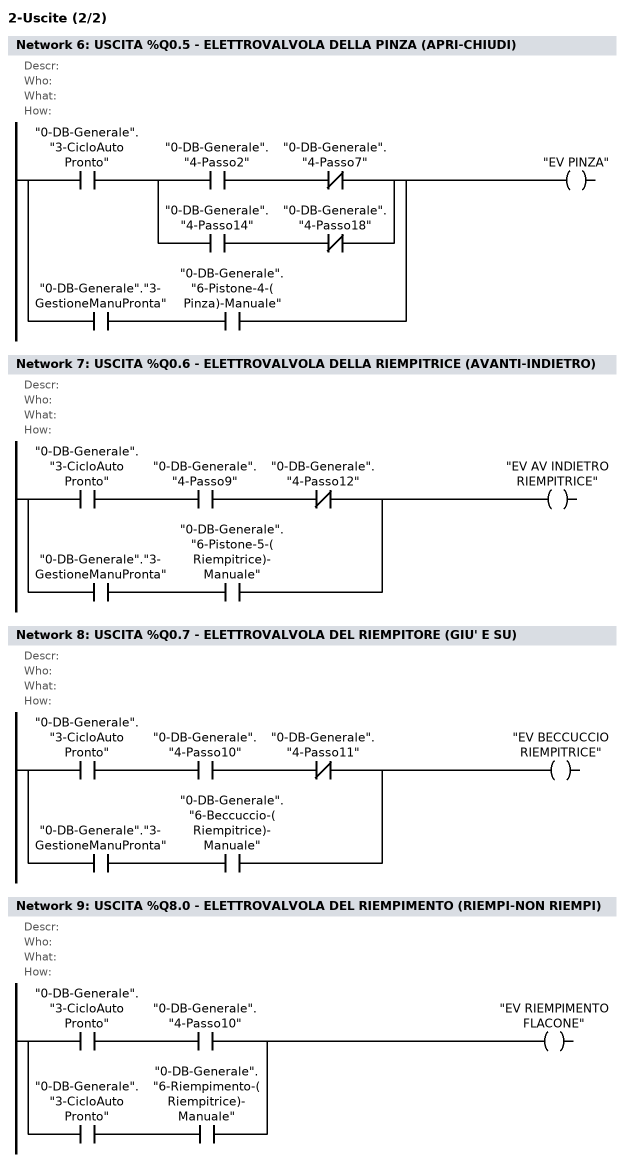
   RUNG wire#powerrail
      Contact( "0-DB-Generale"."3-CicloAutoPronto" )
      wire#w1
      Contact( "0-DB-Generale"."4-Passo2" )
      I_Contact( "0-DB-Generale"."4-Passo7" )
      wire#w2
      Coil( "EV PINZA" )
   END_RUNG
   RUNG wire#w1
      Contact( "0-DB-Generale"."4-Passo14" )
      I_Contact( "0-DB-Generale"."4-Passo18" )
   END_RUNG wire#w2
   RUNG wire#powerrail
      Contact( "0-DB-Generale"."3-GestioneManuPronta" )
      Contact( "0-DB-Generale"."6-Pistone-4-(Pinza)-Manuale" )
   END_RUNG wire#w2
   // the same network as SCL:
   "EV PINZA" := ("0-DB-Generale"."3-CicloAutoPronto" AND (("0-DB-Generale"."4-Passo2" AND NOT "0-DB-Generale"."4-Passo7") OR ("0-DB-Generale"."4-Passo14" AND NOT "0-DB-Generale"."4-Passo18"))) OR ("0-DB-Generale"."3-GestioneManuPronta" AND "0-DB-Generale"."6-Pistone-4-(Pinza)-Manuale");
END_REGION

REGION Network 7: USCITA %Q0.6 - ELETTROVALVOLA DELLA RIEMPITRICE (AVANTI-INDIETRO)
   // Descr: 
   // Who: 
   // What: 
   // How:
   RUNG wire#powerrail
      Contact( "0-DB-Generale"."3-CicloAutoPronto" )
      Contact( "0-DB-Generale"."4-Passo9" )
      I_Contact( "0-DB-Generale"."4-Passo12" )
      wire#w1
      Coil( "EV AV INDIETRO RIEMPITRICE" )
   END_RUNG
   RUNG wire#powerrail
      Contact( "0-DB-Generale"."3-GestioneManuPronta" )
      Contact( "0-DB-Generale"."6-Pistone-5-(Riempitrice)-Manuale" )
   END_RUNG wire#w1
   // the same network as SCL:
   "EV AV INDIETRO RIEMPITRICE" := ("0-DB-Generale"."3-CicloAutoPronto" AND "0-DB-Generale"."4-Passo9" AND NOT "0-DB-Generale"."4-Passo12") OR ("0-DB-Generale"."3-GestioneManuPronta" AND "0-DB-Generale"."6-Pistone-5-(Riempitrice)-Manuale");
END_REGION

REGION Network 8: USCITA %Q0.7 - ELETTROVALVOLA DEL RIEMPITORE (GIU' E SU)
   // Descr: 
   // Who: 
   // What: 
   // How:
   RUNG wire#powerrail
      Contact( "0-DB-Generale"."3-CicloAutoPronto" )
      Contact( "0-DB-Generale"."4-Passo10" )
      I_Contact( "0-DB-Generale"."4-Passo11" )
      wire#w1
      Coil( "EV BECCUCCIO RIEMPITRICE" )
   END_RUNG
   RUNG wire#powerrail
      Contact( "0-DB-Generale"."3-GestioneManuPronta" )
      Contact( "0-DB-Generale"."6-Beccuccio-(Riempitrice)-Manuale" )
   END_RUNG wire#w1
   // the same network as SCL:
   "EV BECCUCCIO RIEMPITRICE" := ("0-DB-Generale"."3-CicloAutoPronto" AND "0-DB-Generale"."4-Passo10" AND NOT "0-DB-Generale"."4-Passo11") OR ("0-DB-Generale"."3-GestioneManuPronta" AND "0-DB-Generale"."6-Beccuccio-(Riempitrice)-Manuale");
END_REGION

REGION Network 9: USCITA %Q8.0 - ELETTROVALVOLA DEL RIEMPIMENTO (RIEMPI-NON RIEMPI)
   // Descr: 
   // Who: 
   // What: 
   // How:
   RUNG wire#powerrail
      Contact( "0-DB-Generale"."3-CicloAutoPronto" )
      Contact( "0-DB-Generale"."4-Passo10" )
      wire#w1
      Coil( "EV RIEMPIMENTO FLACONE" )
   END_RUNG
   RUNG wire#powerrail
      Contact( "0-DB-Generale"."3-CicloAutoPronto" )
      Contact( "0-DB-Generale"."6-Riempimento-(Riempitrice)-Manuale" )
   END_RUNG wire#w1
   // the same network as SCL:
   "EV RIEMPIMENTO FLACONE" := ("0-DB-Generale"."3-CicloAutoPronto" AND "0-DB-Generale"."4-Passo10") OR ("0-DB-Generale"."3-CicloAutoPronto" AND "0-DB-Generale"."6-Riempimento-(Riempitrice)-Manuale");
END_REGION
END_FUNCTION

FUNCTION "3-AvvioAutoManu" : Void   // FC4, LAD
TITLE = NETWORK 1-3: AVVIO CICLO AUTOMATICO; NETWORK 4-5: AVVIO GESTIONE MANUALE
{ S7_Optimized_Access := 'TRUE' }
VERSION : 0.1
BEGIN

REGION Network 1: CONTROLLO SE L'AUTOMAZIONE E' PRONTA AD AVVIARE IL CICLO AUTOMATICO
   // Se la macchina non è in emergenza E il selettore Manu/Auto è in Automatico allora la macchina è pronta per avviare il ciclo automatico
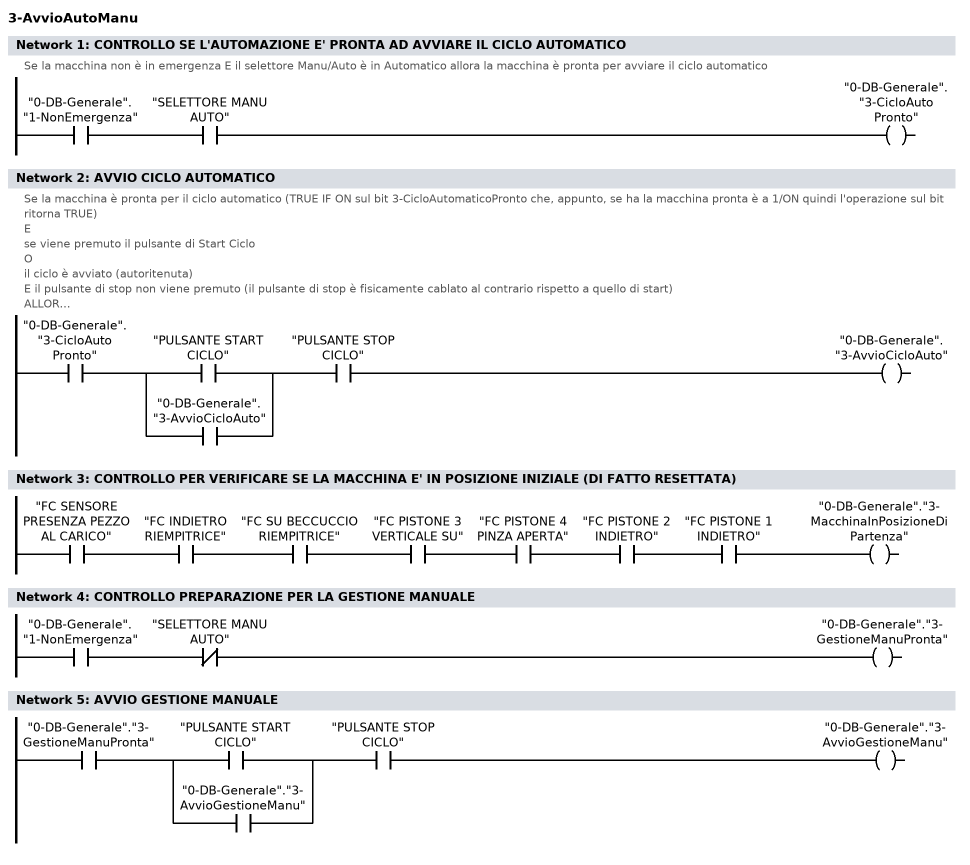
   RUNG wire#powerrail
      Contact( "0-DB-Generale"."1-NonEmergenza" )
      Contact( "SELETTORE MANU  AUTO" )
      Coil( "0-DB-Generale"."3-CicloAutoPronto" )
   END_RUNG
   // the same network as SCL:
   "0-DB-Generale"."3-CicloAutoPronto" := "0-DB-Generale"."1-NonEmergenza" AND "SELETTORE MANU  AUTO";
END_REGION

REGION Network 2: AVVIO CICLO AUTOMATICO
   // Se la macchina è pronta per il ciclo automatico (TRUE IF ON sul bit 3-CicloAutomaticoPronto che, appunto, se ha la macchina pronta è a 1/ON quindi l'operazione sul bit ritorna TRUE) 
   // E 
   // se viene premuto il pulsante di Start Ciclo 
   // O 
   // il ciclo è avviato (autoritenuta) 
   // E il pulsante di stop non viene premuto (il pulsante di stop è fisicamente cablato al contrario rispetto a quello di start) 
   // ALLORA
   // il ciclo automatico si può avviare
   RUNG wire#powerrail
      Contact( "0-DB-Generale"."3-CicloAutoPronto" )
      wire#w1
      Contact( "PULSANTE START CICLO" )
      wire#w2
      Contact( "PULSANTE STOP CICLO" )
      Coil( "0-DB-Generale"."3-AvvioCicloAuto" )
   END_RUNG
   RUNG wire#w1
      Contact( "0-DB-Generale"."3-AvvioCicloAuto" )
   END_RUNG wire#w2
   // the same network as SCL:
   "0-DB-Generale"."3-AvvioCicloAuto" := "0-DB-Generale"."3-CicloAutoPronto" AND ("PULSANTE START CICLO" OR "0-DB-Generale"."3-AvvioCicloAuto") AND "PULSANTE STOP CICLO";
END_REGION

REGION Network 3: CONTROLLO PER VERIFICARE SE LA MACCHINA E' IN POSIZIONE INIZIALE (DI FATTO RESETTATA)
   RUNG wire#powerrail
      Contact( "FC SENSORE PRESENZA PEZZO AL CARICO" )
      Contact( "FC INDIETRO RIEMPITRICE" )
      Contact( "FC SU BECCUCCIO RIEMPITRICE" )
      Contact( "FC PISTONE 3 VERTICALE SU" )
      Contact( "FC PISTONE 4 PINZA APERTA" )
      Contact( "FC PISTONE 2 INDIETRO" )
      Contact( "FC PISTONE 1 INDIETRO" )
      Coil( "0-DB-Generale"."3-MacchinaInPosizioneDiPartenza" )
   END_RUNG
   // the same network as SCL:
   "0-DB-Generale"."3-MacchinaInPosizioneDiPartenza" := "FC SENSORE PRESENZA PEZZO AL CARICO" AND "FC INDIETRO RIEMPITRICE" AND "FC SU BECCUCCIO RIEMPITRICE" AND "FC PISTONE 3 VERTICALE SU" AND "FC PISTONE 4 PINZA APERTA" AND "FC PISTONE 2 INDIETRO" AND "FC PISTONE 1 INDIETRO";
END_REGION

REGION Network 4: CONTROLLO PREPARAZIONE PER LA GESTIONE MANUALE
   RUNG wire#powerrail
      Contact( "0-DB-Generale"."1-NonEmergenza" )
      I_Contact( "SELETTORE MANU  AUTO" )
      Coil( "0-DB-Generale"."3-GestioneManuPronta" )
   END_RUNG
   // the same network as SCL:
   "0-DB-Generale"."3-GestioneManuPronta" := "0-DB-Generale"."1-NonEmergenza" AND NOT "SELETTORE MANU  AUTO";
END_REGION

REGION Network 5: AVVIO GESTIONE MANUALE
   RUNG wire#powerrail
      Contact( "0-DB-Generale"."3-GestioneManuPronta" )
      wire#w1
      Contact( "PULSANTE START CICLO" )
      wire#w2
      Contact( "PULSANTE STOP CICLO" )
      Coil( "0-DB-Generale"."3-AvvioGestioneManu" )
   END_RUNG
   RUNG wire#w1
      Contact( "0-DB-Generale"."3-AvvioGestioneManu" )
   END_RUNG wire#w2
   // the same network as SCL:
   "0-DB-Generale"."3-AvvioGestioneManu" := "0-DB-Generale"."3-GestioneManuPronta" AND ("PULSANTE START CICLO" OR "0-DB-Generale"."3-AvvioGestioneManu") AND "PULSANTE STOP CICLO";
END_REGION
END_FUNCTION

FUNCTION "4-CicloAutomatico" : Void   // FC5, LAD
{ S7_Optimized_Access := 'TRUE' }
VERSION : 0.1
   VAR_TEMP   // added for the SCL form of the ladder/FBD networks
      _w1 : Bool;
   END_VAR
BEGIN

REGION Network 1: Il pistone 3 si abbassa sul flacone (pre riempimento)
   // Se sono presenti tutti i fine corsa come da default (primo rung allora attiva il primo azionamento delle elettrovalvole)
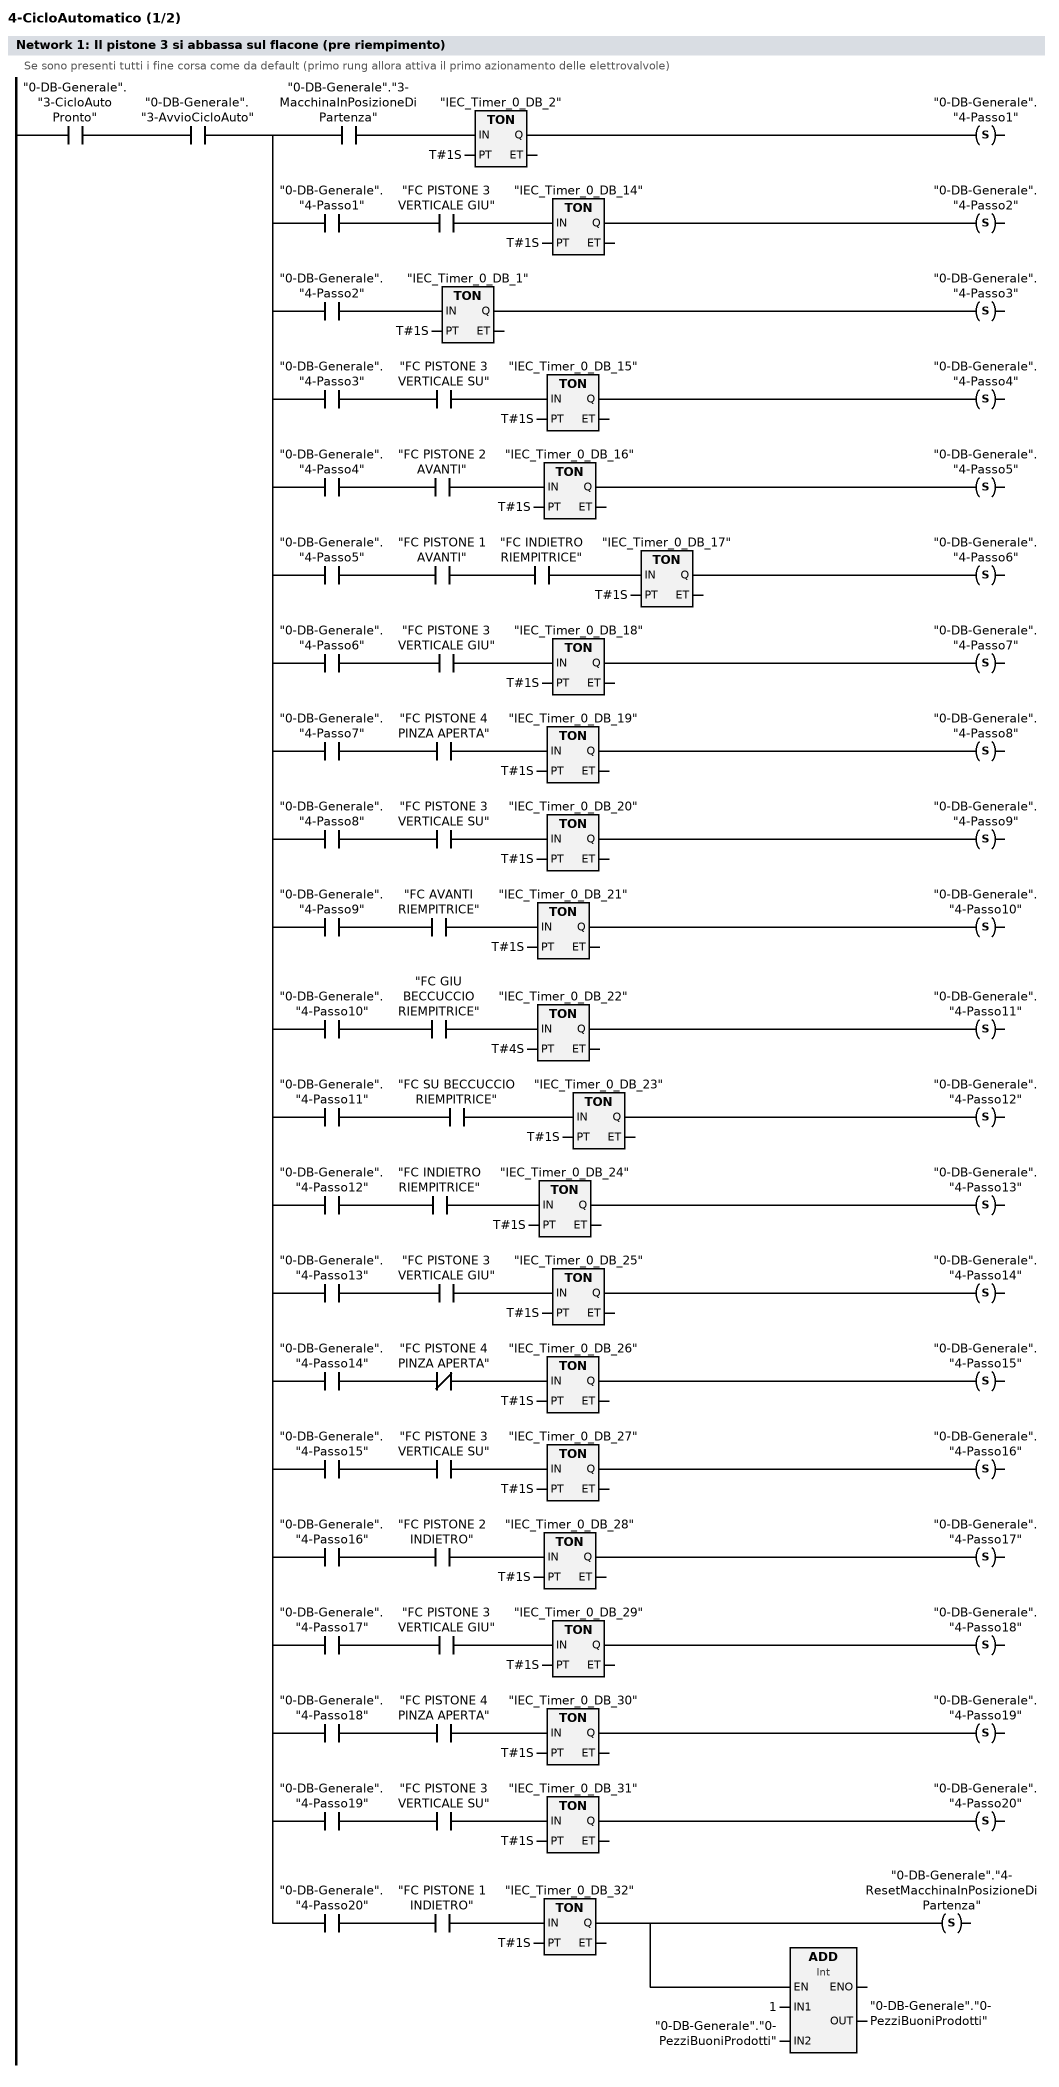
   #_w1 := "0-DB-Generale"."3-CicloAutoPronto" AND "0-DB-Generale"."3-AvvioCicloAuto";
   "IEC_Timer_0_DB_2".TON(IN := #_w1 AND "0-DB-Generale"."3-MacchinaInPosizioneDiPartenza", PT := T#1S);
   IF "IEC_Timer_0_DB_2".Q THEN "0-DB-Generale"."4-Passo1" := TRUE; END_IF;
   "IEC_Timer_0_DB_14".TON(IN := #_w1 AND "0-DB-Generale"."4-Passo1" AND "FC PISTONE 3 VERTICALE GIU",
                           PT := T#1S);
   IF "IEC_Timer_0_DB_14".Q THEN "0-DB-Generale"."4-Passo2" := TRUE; END_IF;
   "IEC_Timer_0_DB_1".TON(IN := #_w1 AND "0-DB-Generale"."4-Passo2", PT := T#1S);
   IF "IEC_Timer_0_DB_1".Q THEN "0-DB-Generale"."4-Passo3" := TRUE; END_IF;
   "IEC_Timer_0_DB_15".TON(IN := #_w1 AND "0-DB-Generale"."4-Passo3" AND "FC PISTONE 3 VERTICALE SU",
                           PT := T#1S);
   IF "IEC_Timer_0_DB_15".Q THEN "0-DB-Generale"."4-Passo4" := TRUE; END_IF;
   "IEC_Timer_0_DB_16".TON(IN := #_w1 AND "0-DB-Generale"."4-Passo4" AND "FC PISTONE 2 AVANTI", PT := T#1S);
   IF "IEC_Timer_0_DB_16".Q THEN "0-DB-Generale"."4-Passo5" := TRUE; END_IF;
   "IEC_Timer_0_DB_17".TON(IN := #_w1 AND "0-DB-Generale"."4-Passo5" AND "FC PISTONE 1 AVANTI" AND "FC INDIETRO RIEMPITRICE",
                           PT := T#1S);
   IF "IEC_Timer_0_DB_17".Q THEN "0-DB-Generale"."4-Passo6" := TRUE; END_IF;
   "IEC_Timer_0_DB_18".TON(IN := #_w1 AND "0-DB-Generale"."4-Passo6" AND "FC PISTONE 3 VERTICALE GIU",
                           PT := T#1S);
   IF "IEC_Timer_0_DB_18".Q THEN "0-DB-Generale"."4-Passo7" := TRUE; END_IF;
   "IEC_Timer_0_DB_19".TON(IN := #_w1 AND "0-DB-Generale"."4-Passo7" AND "FC PISTONE 4 PINZA APERTA",
                           PT := T#1S);
   IF "IEC_Timer_0_DB_19".Q THEN "0-DB-Generale"."4-Passo8" := TRUE; END_IF;
   "IEC_Timer_0_DB_20".TON(IN := #_w1 AND "0-DB-Generale"."4-Passo8" AND "FC PISTONE 3 VERTICALE SU",
                           PT := T#1S);
   IF "IEC_Timer_0_DB_20".Q THEN "0-DB-Generale"."4-Passo9" := TRUE; END_IF;
   "IEC_Timer_0_DB_21".TON(IN := #_w1 AND "0-DB-Generale"."4-Passo9" AND "FC AVANTI RIEMPITRICE", PT := T#1S);
   IF "IEC_Timer_0_DB_21".Q THEN "0-DB-Generale"."4-Passo10" := TRUE; END_IF;
   "IEC_Timer_0_DB_22".TON(IN := #_w1 AND "0-DB-Generale"."4-Passo10" AND "FC GIU BECCUCCIO RIEMPITRICE",
                           PT := T#4S);
   IF "IEC_Timer_0_DB_22".Q THEN "0-DB-Generale"."4-Passo11" := TRUE; END_IF;
   "IEC_Timer_0_DB_23".TON(IN := #_w1 AND "0-DB-Generale"."4-Passo11" AND "FC SU BECCUCCIO RIEMPITRICE",
                           PT := T#1S);
   IF "IEC_Timer_0_DB_23".Q THEN "0-DB-Generale"."4-Passo12" := TRUE; END_IF;
   "IEC_Timer_0_DB_24".TON(IN := #_w1 AND "0-DB-Generale"."4-Passo12" AND "FC INDIETRO RIEMPITRICE", PT := T#1S);
   IF "IEC_Timer_0_DB_24".Q THEN "0-DB-Generale"."4-Passo13" := TRUE; END_IF;
   "IEC_Timer_0_DB_25".TON(IN := #_w1 AND "0-DB-Generale"."4-Passo13" AND "FC PISTONE 3 VERTICALE GIU",
                           PT := T#1S);
   IF "IEC_Timer_0_DB_25".Q THEN "0-DB-Generale"."4-Passo14" := TRUE; END_IF;
   "IEC_Timer_0_DB_26".TON(IN := #_w1 AND "0-DB-Generale"."4-Passo14" AND NOT "FC PISTONE 4 PINZA APERTA",
                           PT := T#1S);
   IF "IEC_Timer_0_DB_26".Q THEN "0-DB-Generale"."4-Passo15" := TRUE; END_IF;
   "IEC_Timer_0_DB_27".TON(IN := #_w1 AND "0-DB-Generale"."4-Passo15" AND "FC PISTONE 3 VERTICALE SU",
                           PT := T#1S);
   IF "IEC_Timer_0_DB_27".Q THEN "0-DB-Generale"."4-Passo16" := TRUE; END_IF;
   "IEC_Timer_0_DB_28".TON(IN := #_w1 AND "0-DB-Generale"."4-Passo16" AND "FC PISTONE 2 INDIETRO", PT := T#1S);
   IF "IEC_Timer_0_DB_28".Q THEN "0-DB-Generale"."4-Passo17" := TRUE; END_IF;
   "IEC_Timer_0_DB_29".TON(IN := #_w1 AND "0-DB-Generale"."4-Passo17" AND "FC PISTONE 3 VERTICALE GIU",
                           PT := T#1S);
   IF "IEC_Timer_0_DB_29".Q THEN "0-DB-Generale"."4-Passo18" := TRUE; END_IF;
   "IEC_Timer_0_DB_30".TON(IN := #_w1 AND "0-DB-Generale"."4-Passo18" AND "FC PISTONE 4 PINZA APERTA",
                           PT := T#1S);
   IF "IEC_Timer_0_DB_30".Q THEN "0-DB-Generale"."4-Passo19" := TRUE; END_IF;
   "IEC_Timer_0_DB_31".TON(IN := #_w1 AND "0-DB-Generale"."4-Passo19" AND "FC PISTONE 3 VERTICALE SU",
                           PT := T#1S);
   IF "IEC_Timer_0_DB_31".Q THEN "0-DB-Generale"."4-Passo20" := TRUE; END_IF;
   "IEC_Timer_0_DB_32".TON(IN := #_w1 AND "0-DB-Generale"."4-Passo20" AND "FC PISTONE 1 INDIETRO", PT := T#1S);
   IF "IEC_Timer_0_DB_32".Q THEN
       "0-DB-Generale"."4-ResetMacchinaInPosizioneDiPartenza" := TRUE;
       "0-DB-Generale"."0-PezziBuoniProdotti" := 1 + "0-DB-Generale"."0-PezziBuoniProdotti";
   END_IF;
END_REGION

REGION Network 2: Il pistone 3 si abbassa sul flacone (pre riempimento)
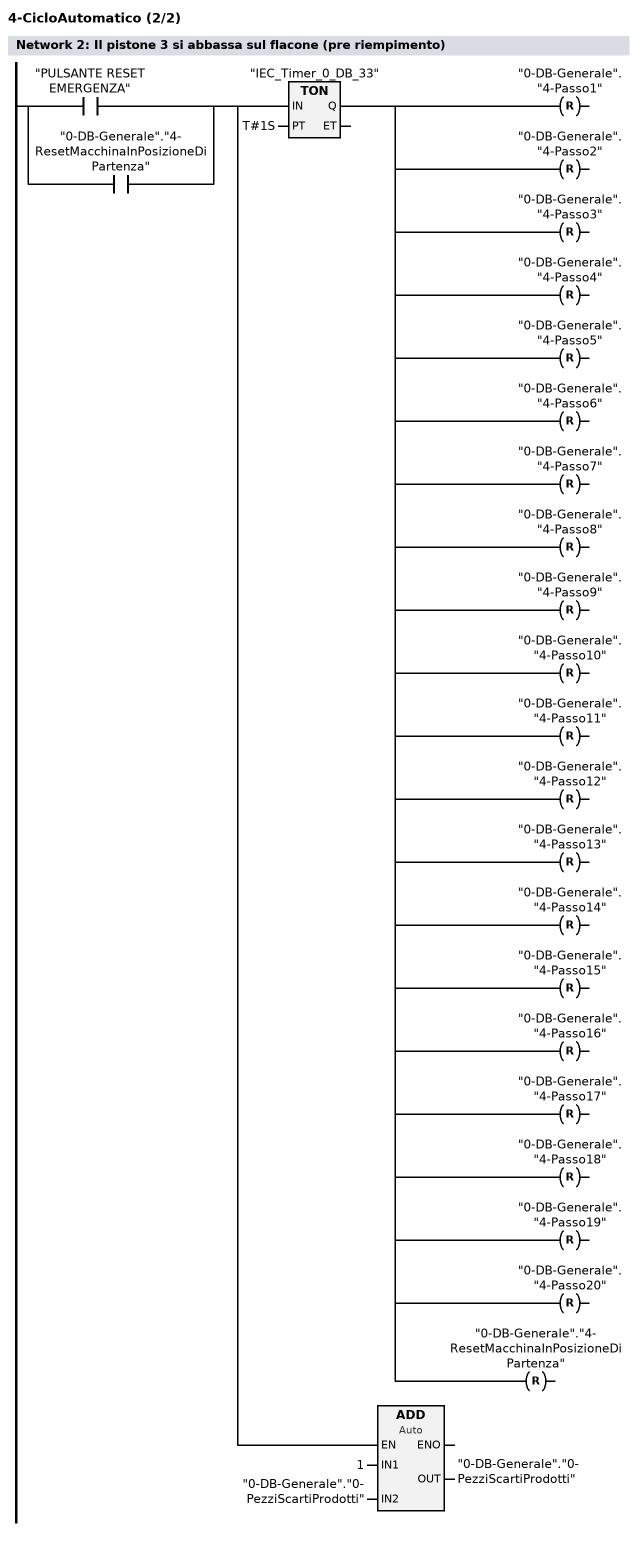
   #_w1 := "PULSANTE RESET EMERGENZA" OR "0-DB-Generale"."4-ResetMacchinaInPosizioneDiPartenza";
   "IEC_Timer_0_DB_33".TON(IN := #_w1, PT := T#1S);
   IF "IEC_Timer_0_DB_33".Q THEN
       "0-DB-Generale"."4-Passo1" := FALSE;
       "0-DB-Generale"."4-Passo2" := FALSE;
       "0-DB-Generale"."4-Passo3" := FALSE;
       "0-DB-Generale"."4-Passo4" := FALSE;
       "0-DB-Generale"."4-Passo5" := FALSE;
       "0-DB-Generale"."4-Passo6" := FALSE;
       "0-DB-Generale"."4-Passo7" := FALSE;
       "0-DB-Generale"."4-Passo8" := FALSE;
       "0-DB-Generale"."4-Passo9" := FALSE;
       "0-DB-Generale"."4-Passo10" := FALSE;
       "0-DB-Generale"."4-Passo11" := FALSE;
       "0-DB-Generale"."4-Passo12" := FALSE;
       "0-DB-Generale"."4-Passo13" := FALSE;
       "0-DB-Generale"."4-Passo14" := FALSE;
       "0-DB-Generale"."4-Passo15" := FALSE;
       "0-DB-Generale"."4-Passo16" := FALSE;
       "0-DB-Generale"."4-Passo17" := FALSE;
       "0-DB-Generale"."4-Passo18" := FALSE;
       "0-DB-Generale"."4-Passo19" := FALSE;
       "0-DB-Generale"."4-Passo20" := FALSE;
       "0-DB-Generale"."4-ResetMacchinaInPosizioneDiPartenza" := FALSE;
   END_IF;
   IF #_w1 THEN
       "0-DB-Generale"."0-PezziScartiProdotti" := 1 + "0-DB-Generale"."0-PezziScartiProdotti";
   END_IF;
END_REGION
END_FUNCTION

FUNCTION "6-CicloManuale" : Void   // FC6, LAD
{ S7_Optimized_Access := 'TRUE' }
VERSION : 0.1
   VAR_TEMP   // added for the SCL form of the ladder/FBD networks
      _w1 : Bool;
   END_VAR
BEGIN

REGION Network 1: GESTIONE DEL PISTONE 1 DI AVANZAMENTO/INDIETREGGIAMENTO DEL MANIPOLATORE
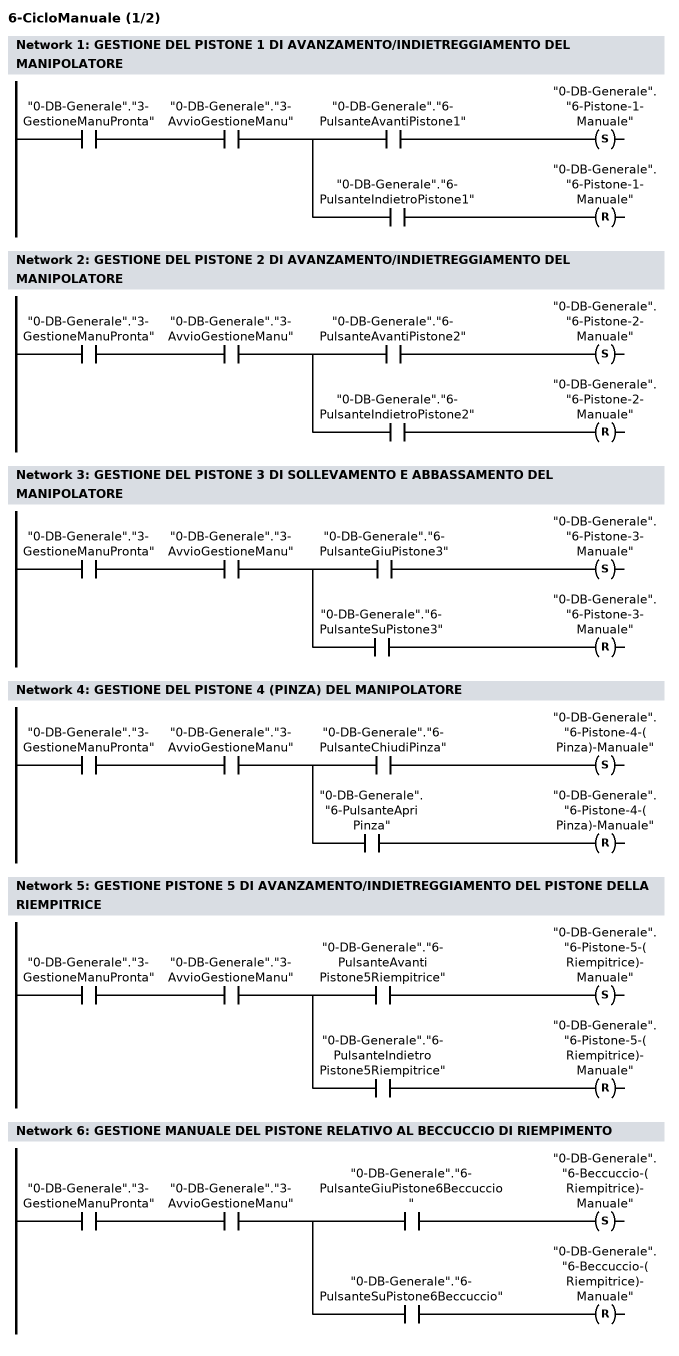
   RUNG wire#powerrail
      Contact( "0-DB-Generale"."3-GestioneManuPronta" )
      Contact( "0-DB-Generale"."3-AvvioGestioneManu" )
      wire#w1
      Contact( "0-DB-Generale"."6-PulsanteAvantiPistone1" )
      S_Coil( "0-DB-Generale"."6-Pistone-1-Manuale" )
   END_RUNG
   RUNG wire#w1
      Contact( "0-DB-Generale"."6-PulsanteIndietroPistone1" )
      R_Coil( "0-DB-Generale"."6-Pistone-1-Manuale" )
   END_RUNG
   // the same network as SCL:
   #_w1 := "0-DB-Generale"."3-GestioneManuPronta" AND "0-DB-Generale"."3-AvvioGestioneManu";
   IF #_w1 AND "0-DB-Generale"."6-PulsanteAvantiPistone1" THEN
       "0-DB-Generale"."6-Pistone-1-Manuale" := TRUE;
   END_IF;
   IF #_w1 AND "0-DB-Generale"."6-PulsanteIndietroPistone1" THEN
       "0-DB-Generale"."6-Pistone-1-Manuale" := FALSE;
   END_IF;
END_REGION

REGION Network 2: GESTIONE DEL PISTONE 2 DI AVANZAMENTO/INDIETREGGIAMENTO DEL MANIPOLATORE
   RUNG wire#powerrail
      Contact( "0-DB-Generale"."3-GestioneManuPronta" )
      Contact( "0-DB-Generale"."3-AvvioGestioneManu" )
      wire#w1
      Contact( "0-DB-Generale"."6-PulsanteAvantiPistone2" )
      S_Coil( "0-DB-Generale"."6-Pistone-2-Manuale" )
   END_RUNG
   RUNG wire#w1
      Contact( "0-DB-Generale"."6-PulsanteIndietroPistone2" )
      R_Coil( "0-DB-Generale"."6-Pistone-2-Manuale" )
   END_RUNG
   // the same network as SCL:
   #_w1 := "0-DB-Generale"."3-GestioneManuPronta" AND "0-DB-Generale"."3-AvvioGestioneManu";
   IF #_w1 AND "0-DB-Generale"."6-PulsanteAvantiPistone2" THEN
       "0-DB-Generale"."6-Pistone-2-Manuale" := TRUE;
   END_IF;
   IF #_w1 AND "0-DB-Generale"."6-PulsanteIndietroPistone2" THEN
       "0-DB-Generale"."6-Pistone-2-Manuale" := FALSE;
   END_IF;
END_REGION

REGION Network 3: GESTIONE DEL PISTONE 3 DI SOLLEVAMENTO E ABBASSAMENTO DEL MANIPOLATORE
   RUNG wire#powerrail
      Contact( "0-DB-Generale"."3-GestioneManuPronta" )
      Contact( "0-DB-Generale"."3-AvvioGestioneManu" )
      wire#w1
      Contact( "0-DB-Generale"."6-PulsanteGiuPistone3" )
      S_Coil( "0-DB-Generale"."6-Pistone-3-Manuale" )
   END_RUNG
   RUNG wire#w1
      Contact( "0-DB-Generale"."6-PulsanteSuPistone3" )
      R_Coil( "0-DB-Generale"."6-Pistone-3-Manuale" )
   END_RUNG
   // the same network as SCL:
   #_w1 := "0-DB-Generale"."3-GestioneManuPronta" AND "0-DB-Generale"."3-AvvioGestioneManu";
   IF #_w1 AND "0-DB-Generale"."6-PulsanteGiuPistone3" THEN
       "0-DB-Generale"."6-Pistone-3-Manuale" := TRUE;
   END_IF;
   IF #_w1 AND "0-DB-Generale"."6-PulsanteSuPistone3" THEN
       "0-DB-Generale"."6-Pistone-3-Manuale" := FALSE;
   END_IF;
END_REGION

REGION Network 4: GESTIONE DEL PISTONE 4 (PINZA) DEL MANIPOLATORE
   RUNG wire#powerrail
      Contact( "0-DB-Generale"."3-GestioneManuPronta" )
      Contact( "0-DB-Generale"."3-AvvioGestioneManu" )
      wire#w1
      Contact( "0-DB-Generale"."6-PulsanteChiudiPinza" )
      S_Coil( "0-DB-Generale"."6-Pistone-4-(Pinza)-Manuale" )
   END_RUNG
   RUNG wire#w1
      Contact( "0-DB-Generale"."6-PulsanteApriPinza" )
      R_Coil( "0-DB-Generale"."6-Pistone-4-(Pinza)-Manuale" )
   END_RUNG
   // the same network as SCL:
   #_w1 := "0-DB-Generale"."3-GestioneManuPronta" AND "0-DB-Generale"."3-AvvioGestioneManu";
   IF #_w1 AND "0-DB-Generale"."6-PulsanteChiudiPinza" THEN
       "0-DB-Generale"."6-Pistone-4-(Pinza)-Manuale" := TRUE;
   END_IF;
   IF #_w1 AND "0-DB-Generale"."6-PulsanteApriPinza" THEN
       "0-DB-Generale"."6-Pistone-4-(Pinza)-Manuale" := FALSE;
   END_IF;
END_REGION

REGION Network 5: GESTIONE PISTONE 5 DI AVANZAMENTO/INDIETREGGIAMENTO DEL PISTONE DELLA RIEMPITRICE
   RUNG wire#powerrail
      Contact( "0-DB-Generale"."3-GestioneManuPronta" )
      Contact( "0-DB-Generale"."3-AvvioGestioneManu" )
      wire#w1
      Contact( "0-DB-Generale"."6-PulsanteAvantiPistone5Riempitrice" )
      S_Coil( "0-DB-Generale"."6-Pistone-5-(Riempitrice)-Manuale" )
   END_RUNG
   RUNG wire#w1
      Contact( "0-DB-Generale"."6-PulsanteIndietroPistone5Riempitrice" )
      R_Coil( "0-DB-Generale"."6-Pistone-5-(Riempitrice)-Manuale" )
   END_RUNG
   // the same network as SCL:
   #_w1 := "0-DB-Generale"."3-GestioneManuPronta" AND "0-DB-Generale"."3-AvvioGestioneManu";
   IF #_w1 AND "0-DB-Generale"."6-PulsanteAvantiPistone5Riempitrice" THEN
       "0-DB-Generale"."6-Pistone-5-(Riempitrice)-Manuale" := TRUE;
   END_IF;
   IF #_w1 AND "0-DB-Generale"."6-PulsanteIndietroPistone5Riempitrice" THEN
       "0-DB-Generale"."6-Pistone-5-(Riempitrice)-Manuale" := FALSE;
   END_IF;
END_REGION

REGION Network 6: GESTIONE MANUALE DEL PISTONE RELATIVO AL BECCUCCIO DI RIEMPIMENTO
   RUNG wire#powerrail
      Contact( "0-DB-Generale"."3-GestioneManuPronta" )
      Contact( "0-DB-Generale"."3-AvvioGestioneManu" )
      wire#w1
      Contact( "0-DB-Generale"."6-PulsanteGiuPistone6Beccuccio" )
      S_Coil( "0-DB-Generale"."6-Beccuccio-(Riempitrice)-Manuale" )
   END_RUNG
   RUNG wire#w1
      Contact( "0-DB-Generale"."6-PulsanteSuPistone6Beccuccio" )
      R_Coil( "0-DB-Generale"."6-Beccuccio-(Riempitrice)-Manuale" )
   END_RUNG
   // the same network as SCL:
   #_w1 := "0-DB-Generale"."3-GestioneManuPronta" AND "0-DB-Generale"."3-AvvioGestioneManu";
   IF #_w1 AND "0-DB-Generale"."6-PulsanteGiuPistone6Beccuccio" THEN
       "0-DB-Generale"."6-Beccuccio-(Riempitrice)-Manuale" := TRUE;
   END_IF;
   IF #_w1 AND "0-DB-Generale"."6-PulsanteSuPistone6Beccuccio" THEN
       "0-DB-Generale"."6-Beccuccio-(Riempitrice)-Manuale" := FALSE;
   END_IF;
END_REGION

REGION Network 7: GESTIONE MANUALE DEL RIEMPIMENTO
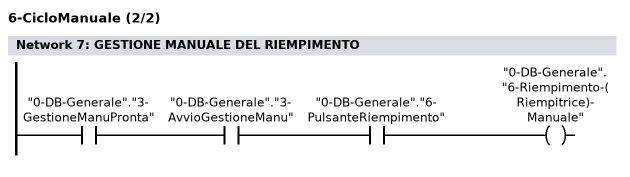
   RUNG wire#powerrail
      Contact( "0-DB-Generale"."3-GestioneManuPronta" )
      Contact( "0-DB-Generale"."3-AvvioGestioneManu" )
      Contact( "0-DB-Generale"."6-PulsanteRiempimento" )
      Coil( "0-DB-Generale"."6-Riempimento-(Riempitrice)-Manuale" )
   END_RUNG
   // the same network as SCL:
   "0-DB-Generale"."6-Riempimento-(Riempitrice)-Manuale" := "0-DB-Generale"."3-GestioneManuPronta" AND "0-DB-Generale"."3-AvvioGestioneManu" AND "0-DB-Generale"."6-PulsanteRiempimento";
END_REGION
END_FUNCTION

FUNCTION "5-HmiUtilities" : Void   // FC7, LAD
{ S7_Optimized_Access := 'TRUE' }
VERSION : 0.1
BEGIN

REGION Network 1: Variabile che gestisce l'obbligo di esecuzione del login: compare un messaggio temporizzato a 5s ogni volta che si cliccano elementi cliccabili nell'HMI senza effettuare il login
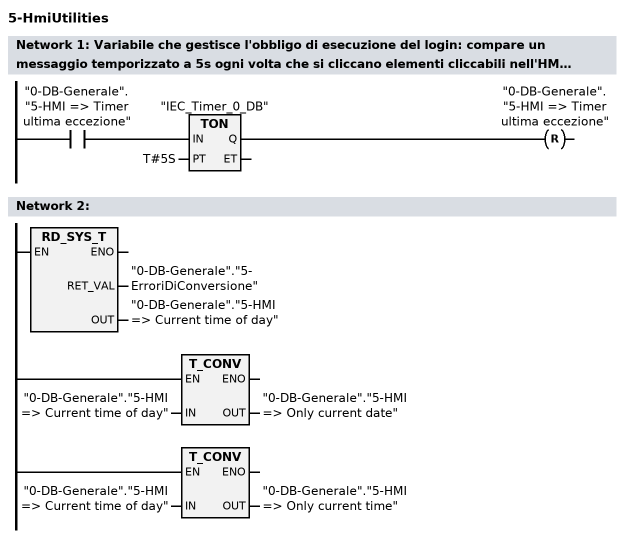
   "IEC_Timer_0_DB".TON(IN := "0-DB-Generale"."5-HMI => Timer ultima eccezione", PT := T#5S);
   IF "IEC_Timer_0_DB".Q THEN "0-DB-Generale"."5-HMI => Timer ultima eccezione" := FALSE; END_IF;
END_REGION

REGION Network 2
   "0-DB-Generale"."5-ErroriDiConversione" := RD_SYS_T(OUT => "0-DB-Generale"."5-HMI => Current time of day");
   "0-DB-Generale"."5-HMI => Only current date" := T_CONV(IN := "0-DB-Generale"."5-HMI => Current time of day");
   "0-DB-Generale"."5-HMI => Only current time" := T_CONV(IN := "0-DB-Generale"."5-HMI => Current time of day");
END_REGION
END_FUNCTION

ORGANIZATION_BLOCK "Main"   // OB1, LAD, ProgramCycle
TITLE = "Main Program Sweep (Cycle)"
{ S7_Optimized_Access := 'TRUE' }
VERSION : 0.1
   VAR_INPUT
      Initial_Call : Bool;   // Initial call of this OB
      Remanence : Bool;   // =True, if remanent data are available
   END_VAR
   VAR_TEMP   // added for the SCL form of the ladder/FBD networks
      _w1 : Bool;
      _w2 : Bool;
      _w3 : Bool;
      _w4 : Bool;
      _w5 : Bool;
   END_VAR
BEGIN

REGION Network 1: GESTIONE SIMULATORE
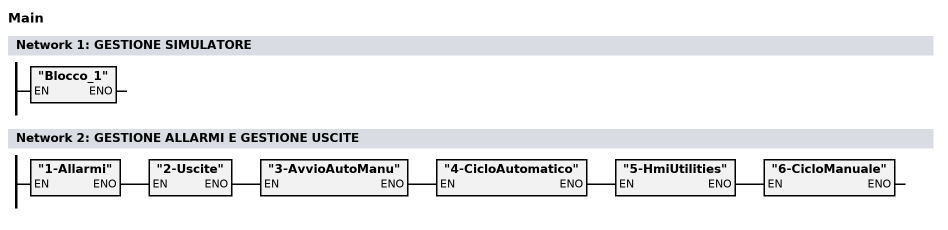
   RUNG wire#powerrail
      "Blocco_1"()
   END_RUNG
   // the same network as SCL:
   "Blocco_1"();
END_REGION

REGION Network 2: GESTIONE ALLARMI E GESTIONE USCITE
   RUNG wire#powerrail
      "1-Allarmi"()
      "2-Uscite"()
      "3-AvvioAutoManu"()
      "4-CicloAutomatico"()
      "5-HmiUtilities"()
      "6-CicloManuale"()
   END_RUNG
   // the same network as SCL:
   "1-Allarmi"(ENO => #_w1);
   "2-Uscite"(EN := #_w1, ENO => #_w2);
   "3-AvvioAutoManu"(EN := #_w2, ENO => #_w3);
   "4-CicloAutomatico"(EN := #_w3, ENO => #_w4);
   "5-HmiUtilities"(EN := #_w4, ENO => #_w5);
   IF #_w5 THEN "6-CicloManuale"(); END_IF;
END_REGION

REGION Network 3: CICLO AUTOMATICO
END_REGION

REGION Network 4: CICLO MANUALE
END_REGION
END_ORGANIZATION_BLOCK

// folder: RISERVATO_NON_MODIFICARE

FUNCTION "Blocco_1" : Void   // FC1, LAD
{ S7_Optimized_Access := 'TRUE' }
VERSION : 0.1
   VAR_TEMP   // added for the SCL form of the ladder/FBD networks
      _w1 : Bool;
      _w2 : Bool;
      _w3 : Bool;
   END_VAR
BEGIN

REGION Network 1: comando pistone 1 prima misura
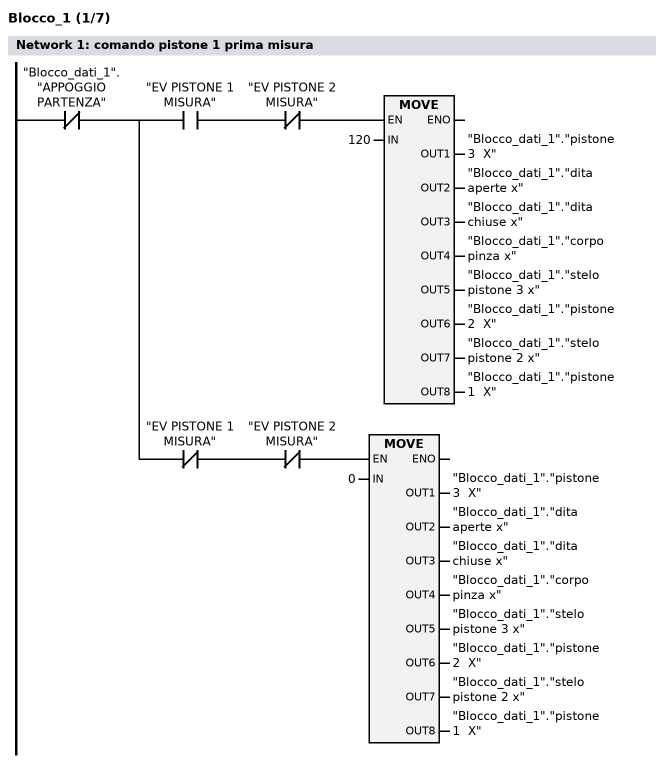
   RUNG wire#powerrail
      I_Contact( "Blocco_dati_1"."APPOGGIO PARTENZA" )
      wire#w1
      Contact( "EV PISTONE 1 MISURA" )
      I_Contact( "EV PISTONE 2 MISURA" )
      Move(in := 120, out1 => "Blocco_dati_1"."pistone 3  X", out2 => "Blocco_dati_1"."dita aperte x", out3 => "Blocco_dati_1"."dita chiuse x", out4 => "Blocco_dati_1"."corpo pinza x", out5 => "Blocco_dati_1"."stelo pistone 3 x", out6 => "Blocco_dati_1"."pistone 2  X", out7 => "Blocco_dati_1"."stelo pistone 2 x", out8 => "Blocco_dati_1"."pistone 1  X")
   END_RUNG
   RUNG wire#w1
      I_Contact( "EV PISTONE 1 MISURA" )
      I_Contact( "EV PISTONE 2 MISURA" )
      Move(in := 0, out1 => "Blocco_dati_1"."pistone 3  X", out2 => "Blocco_dati_1"."dita aperte x", out3 => "Blocco_dati_1"."dita chiuse x", out4 => "Blocco_dati_1"."corpo pinza x", out5 => "Blocco_dati_1"."stelo pistone 3 x", out6 => "Blocco_dati_1"."pistone 2  X", out7 => "Blocco_dati_1"."stelo pistone 2 x", out8 => "Blocco_dati_1"."pistone 1  X")
   END_RUNG
   // the same network as SCL:
   #_w1 := NOT "Blocco_dati_1"."APPOGGIO PARTENZA";
   IF #_w1 AND "EV PISTONE 1 MISURA" AND NOT "EV PISTONE 2 MISURA" THEN
       "Blocco_dati_1"."pistone 3  X" := 120;
       "Blocco_dati_1"."dita aperte x" := 120;
       "Blocco_dati_1"."dita chiuse x" := 120;
       "Blocco_dati_1"."corpo pinza x" := 120;
       "Blocco_dati_1"."stelo pistone 3 x" := 120;
       "Blocco_dati_1"."pistone 2  X" := 120;
       "Blocco_dati_1"."stelo pistone 2 x" := 120;
       "Blocco_dati_1"."pistone 1  X" := 120;
   END_IF;
   IF #_w1 AND NOT "EV PISTONE 1 MISURA" AND NOT "EV PISTONE 2 MISURA" THEN
       "Blocco_dati_1"."pistone 3  X" := 0;
       "Blocco_dati_1"."dita aperte x" := 0;
       "Blocco_dati_1"."dita chiuse x" := 0;
       "Blocco_dati_1"."corpo pinza x" := 0;
       "Blocco_dati_1"."stelo pistone 3 x" := 0;
       "Blocco_dati_1"."pistone 2  X" := 0;
       "Blocco_dati_1"."stelo pistone 2 x" := 0;
       "Blocco_dati_1"."pistone 1  X" := 0;
   END_IF;
END_REGION

REGION Network 2: comando pistone 1 prima misura 120 / SECONDA MISURA = 240
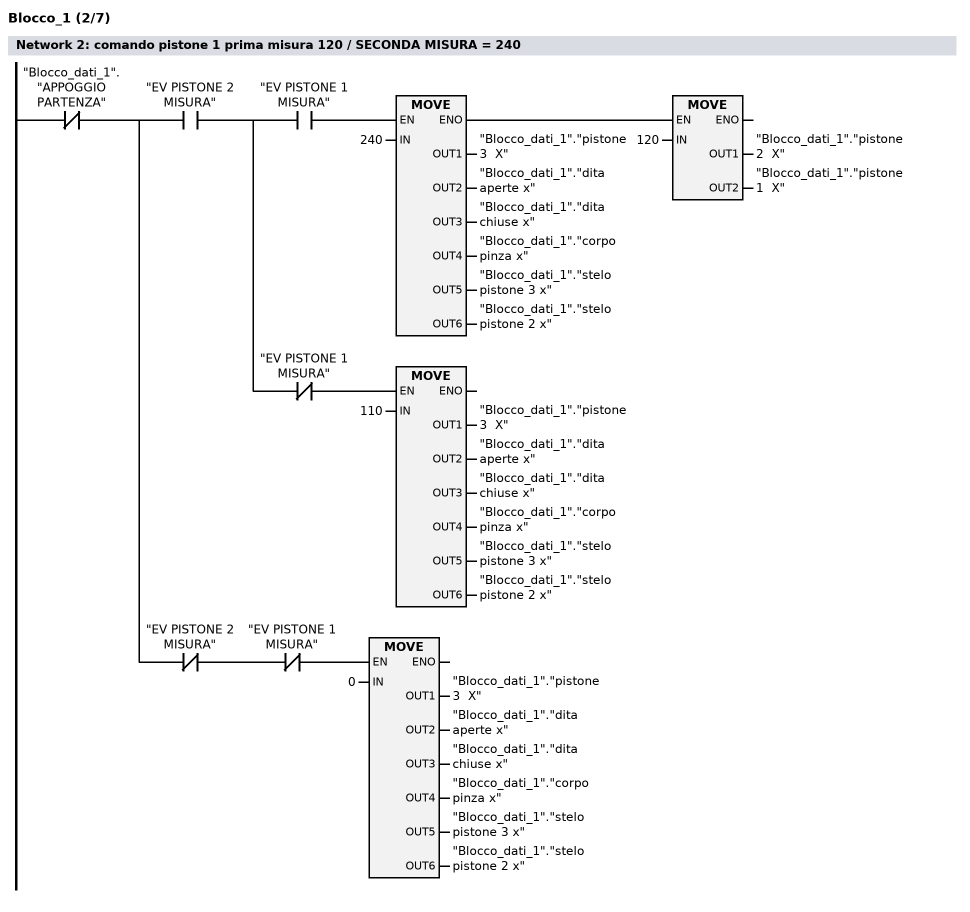
   RUNG wire#powerrail
      I_Contact( "Blocco_dati_1"."APPOGGIO PARTENZA" )
      wire#w1
      Contact( "EV PISTONE 2 MISURA" )
      wire#w2
      Contact( "EV PISTONE 1 MISURA" )
      Move(in := 240, out1 => "Blocco_dati_1"."pistone 3  X", out2 => "Blocco_dati_1"."dita aperte x", out3 => "Blocco_dati_1"."dita chiuse x", out4 => "Blocco_dati_1"."corpo pinza x", out5 => "Blocco_dati_1"."stelo pistone 3 x", out6 => "Blocco_dati_1"."stelo pistone 2 x")
      Move(in := 120, out1 => "Blocco_dati_1"."pistone 2  X", out2 => "Blocco_dati_1"."pistone 1  X")
   END_RUNG
   RUNG wire#w2
      I_Contact( "EV PISTONE 1 MISURA" )
      Move(in := 110, out1 => "Blocco_dati_1"."pistone 3  X", out2 => "Blocco_dati_1"."dita aperte x", out3 => "Blocco_dati_1"."dita chiuse x", out4 => "Blocco_dati_1"."corpo pinza x", out5 => "Blocco_dati_1"."stelo pistone 3 x", out6 => "Blocco_dati_1"."stelo pistone 2 x")
   END_RUNG
   RUNG wire#w1
      I_Contact( "EV PISTONE 2 MISURA" )
      I_Contact( "EV PISTONE 1 MISURA" )
      Move(in := 0, out1 => "Blocco_dati_1"."pistone 3  X", out2 => "Blocco_dati_1"."dita aperte x", out3 => "Blocco_dati_1"."dita chiuse x", out4 => "Blocco_dati_1"."corpo pinza x", out5 => "Blocco_dati_1"."stelo pistone 3 x", out6 => "Blocco_dati_1"."stelo pistone 2 x")
   END_RUNG
   // the same network as SCL:
   #_w1 := NOT "Blocco_dati_1"."APPOGGIO PARTENZA";
   #_w2 := #_w1 AND "EV PISTONE 2 MISURA";
   IF #_w2 AND "EV PISTONE 1 MISURA" THEN
       "Blocco_dati_1"."pistone 3  X" := 240;
       "Blocco_dati_1"."dita aperte x" := 240;
       "Blocco_dati_1"."dita chiuse x" := 240;
       "Blocco_dati_1"."corpo pinza x" := 240;
       "Blocco_dati_1"."stelo pistone 3 x" := 240;
       "Blocco_dati_1"."stelo pistone 2 x" := 240;
       "Blocco_dati_1"."pistone 2  X" := 120;
       "Blocco_dati_1"."pistone 1  X" := 120;
   END_IF;
   IF #_w2 AND NOT "EV PISTONE 1 MISURA" THEN
       "Blocco_dati_1"."pistone 3  X" := 110;
       "Blocco_dati_1"."dita aperte x" := 110;
       "Blocco_dati_1"."dita chiuse x" := 110;
       "Blocco_dati_1"."corpo pinza x" := 110;
       "Blocco_dati_1"."stelo pistone 3 x" := 110;
       "Blocco_dati_1"."stelo pistone 2 x" := 110;
   END_IF;
   IF #_w1 AND NOT "EV PISTONE 2 MISURA" AND NOT "EV PISTONE 1 MISURA" THEN
       "Blocco_dati_1"."pistone 3  X" := 0;
       "Blocco_dati_1"."dita aperte x" := 0;
       "Blocco_dati_1"."dita chiuse x" := 0;
       "Blocco_dati_1"."corpo pinza x" := 0;
       "Blocco_dati_1"."stelo pistone 3 x" := 0;
       "Blocco_dati_1"."stelo pistone 2 x" := 0;
   END_IF;
END_REGION

REGION Network 3: pinza SU GIU PINZA = 90
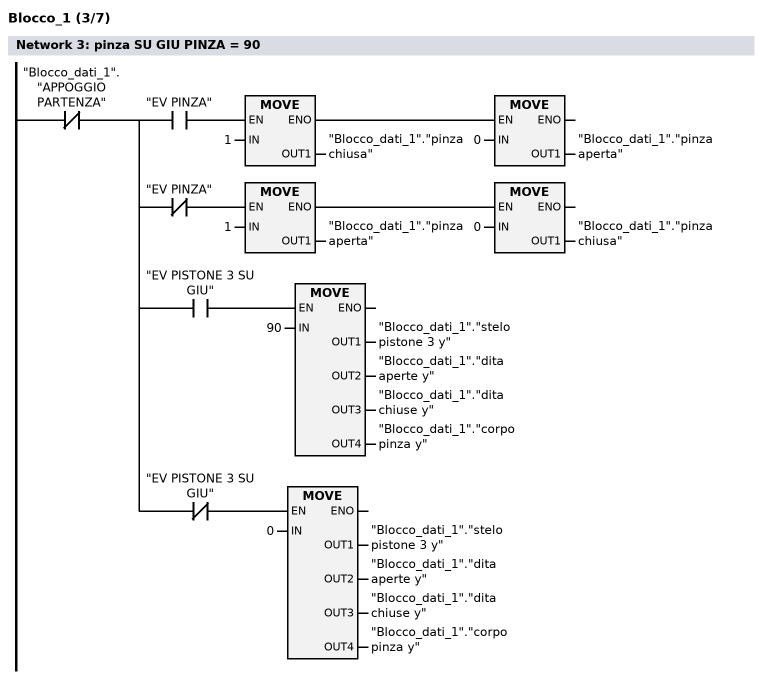
   RUNG wire#powerrail
      I_Contact( "Blocco_dati_1"."APPOGGIO PARTENZA" )
      wire#w1
      Contact( "EV PINZA" )
      Move(in := 1, out1 => "Blocco_dati_1"."pinza chiusa")
      Move(in := 0, out1 => "Blocco_dati_1"."pinza aperta")
   END_RUNG
   RUNG wire#w1
      I_Contact( "EV PINZA" )
      Move(in := 1, out1 => "Blocco_dati_1"."pinza aperta")
      Move(in := 0, out1 => "Blocco_dati_1"."pinza chiusa")
   END_RUNG
   RUNG wire#w1
      Contact( "EV PISTONE 3 SU GIU" )
      Move(in := 90, out1 => "Blocco_dati_1"."stelo pistone 3 y", out2 => "Blocco_dati_1"."dita aperte y", out3 => "Blocco_dati_1"."dita chiuse y", out4 => "Blocco_dati_1"."corpo pinza y")
   END_RUNG
   RUNG wire#w1
      I_Contact( "EV PISTONE 3 SU GIU" )
      Move(in := 0, out1 => "Blocco_dati_1"."stelo pistone 3 y", out2 => "Blocco_dati_1"."dita aperte y", out3 => "Blocco_dati_1"."dita chiuse y", out4 => "Blocco_dati_1"."corpo pinza y")
   END_RUNG
   // the same network as SCL:
   #_w1 := NOT "Blocco_dati_1"."APPOGGIO PARTENZA";
   IF #_w1 AND "EV PINZA" THEN
       "Blocco_dati_1"."pinza chiusa" := 1;
       "Blocco_dati_1"."pinza aperta" := 0;
   END_IF;
   IF #_w1 AND NOT "EV PINZA" THEN
       "Blocco_dati_1"."pinza aperta" := 1;
       "Blocco_dati_1"."pinza chiusa" := 0;
   END_IF;
   IF #_w1 AND "EV PISTONE 3 SU GIU" THEN
       "Blocco_dati_1"."stelo pistone 3 y" := 90;
       "Blocco_dati_1"."dita aperte y" := 90;
       "Blocco_dati_1"."dita chiuse y" := 90;
       "Blocco_dati_1"."corpo pinza y" := 90;
   END_IF;
   IF #_w1 AND NOT "EV PISTONE 3 SU GIU" THEN
       "Blocco_dati_1"."stelo pistone 3 y" := 0;
       "Blocco_dati_1"."dita aperte y" := 0;
       "Blocco_dati_1"."dita chiuse y" := 0;
       "Blocco_dati_1"."corpo pinza y" := 0;
   END_IF;
END_REGION

REGION Network 4: pezzo -90
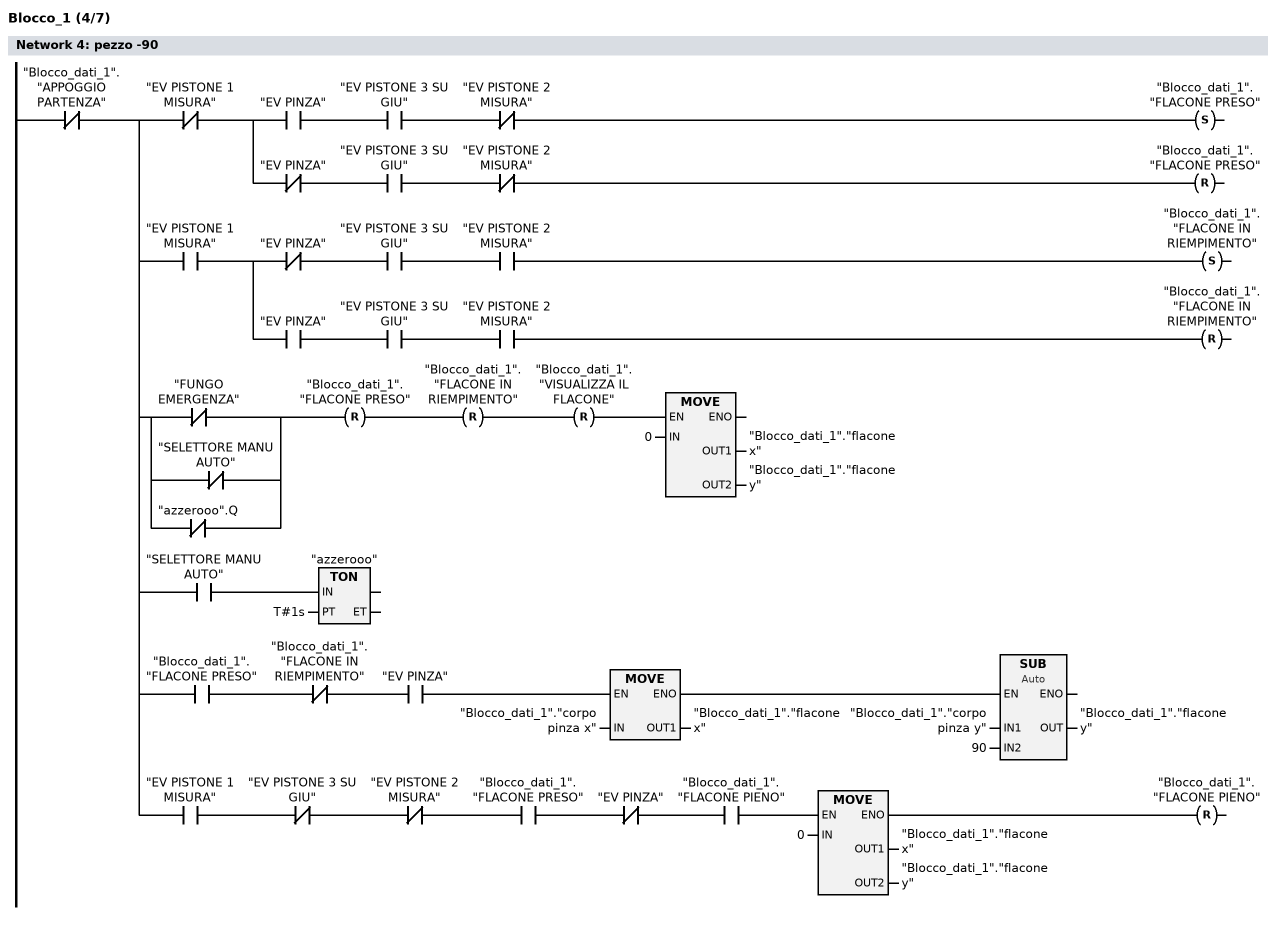
   #_w1 := NOT "Blocco_dati_1"."APPOGGIO PARTENZA";
   #_w2 := #_w1 AND NOT "EV PISTONE 1 MISURA";
   IF #_w2 AND "EV PINZA" AND "EV PISTONE 3 SU GIU" AND NOT "EV PISTONE 2 MISURA" THEN
       "Blocco_dati_1"."FLACONE PRESO" := TRUE;
   END_IF;
   IF #_w2 AND NOT "EV PINZA" AND "EV PISTONE 3 SU GIU" AND NOT "EV PISTONE 2 MISURA" THEN
       "Blocco_dati_1"."FLACONE PRESO" := FALSE;
   END_IF;
   #_w3 := #_w1 AND "EV PISTONE 1 MISURA";
   IF #_w3 AND NOT "EV PINZA" AND "EV PISTONE 3 SU GIU" AND "EV PISTONE 2 MISURA" THEN
       "Blocco_dati_1"."FLACONE IN RIEMPIMENTO" := TRUE;
   END_IF;
   IF #_w3 AND "EV PINZA" AND "EV PISTONE 3 SU GIU" AND "EV PISTONE 2 MISURA" THEN
       "Blocco_dati_1"."FLACONE IN RIEMPIMENTO" := FALSE;
   END_IF;
   IF #_w1 AND (NOT "FUNGO EMERGENZA" OR NOT "SELETTORE MANU  AUTO" OR NOT "azzerooo".Q) THEN
       "Blocco_dati_1"."FLACONE PRESO" := FALSE;
       "Blocco_dati_1"."FLACONE IN RIEMPIMENTO" := FALSE;
       "Blocco_dati_1"."VISUALIZZA IL FLACONE" := FALSE;
       "Blocco_dati_1"."flacone x" := 0;
       "Blocco_dati_1"."flacone y" := 0;
   END_IF;
   "azzerooo".TON(IN := #_w1 AND "SELETTORE MANU  AUTO", PT := T#1s);
   IF #_w1 AND "Blocco_dati_1"."FLACONE PRESO" AND NOT "Blocco_dati_1"."FLACONE IN RIEMPIMENTO" AND "EV PINZA" THEN
       "Blocco_dati_1"."flacone x" := "Blocco_dati_1"."corpo pinza x";
       "Blocco_dati_1"."flacone y" := "Blocco_dati_1"."corpo pinza y" - 90;
   END_IF;
   IF #_w1 AND "EV PISTONE 1 MISURA" AND NOT "EV PISTONE 3 SU GIU" AND NOT "EV PISTONE 2 MISURA" AND "Blocco_dati_1"."FLACONE PRESO" AND NOT "EV PINZA" AND "Blocco_dati_1"."FLACONE PIENO" THEN
       "Blocco_dati_1"."flacone x" := 0;
       "Blocco_dati_1"."flacone y" := 0;
       "Blocco_dati_1"."FLACONE PIENO" := FALSE;
   END_IF;
END_REGION

REGION Network 5: comando riempitrice -90
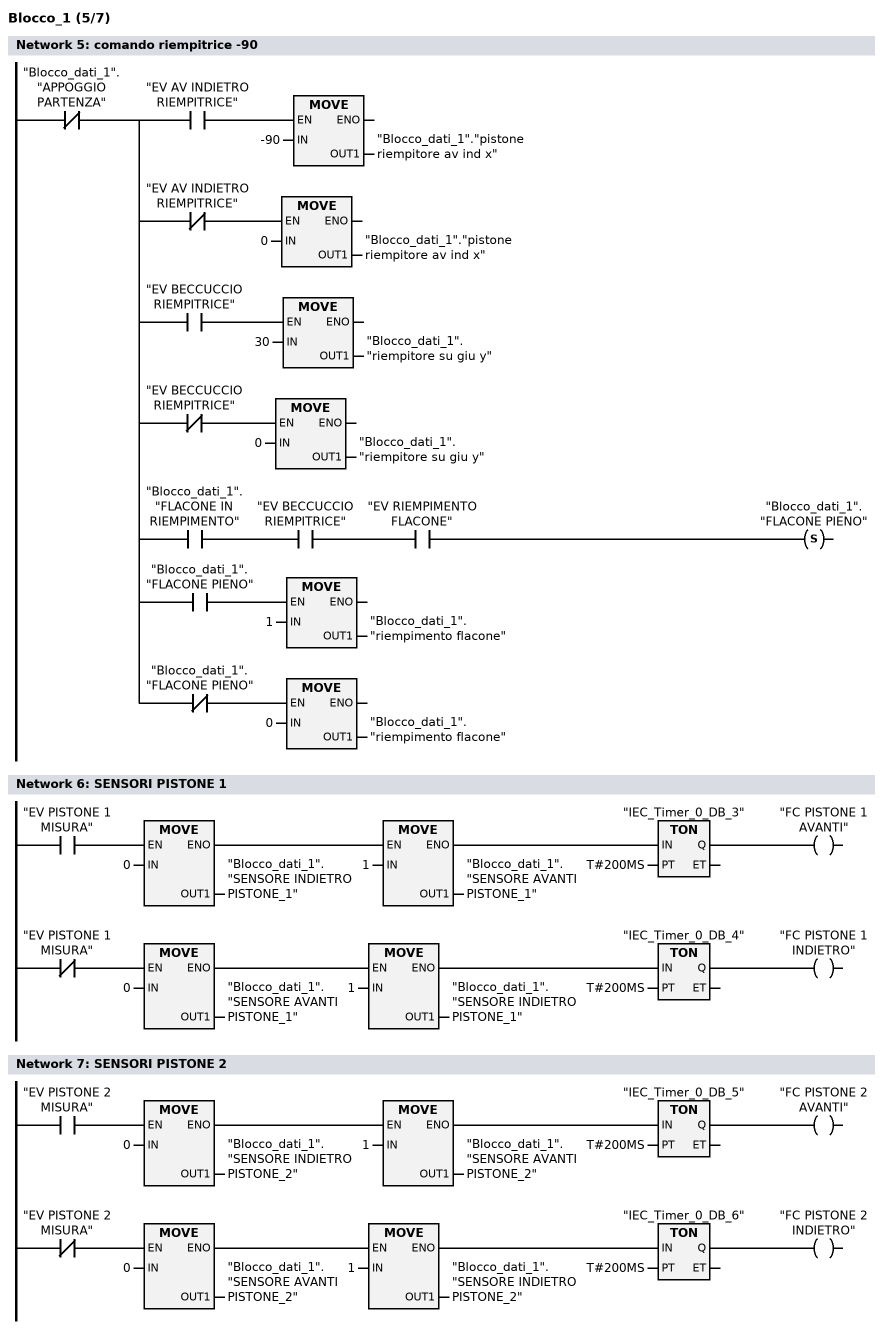
   RUNG wire#powerrail
      I_Contact( "Blocco_dati_1"."APPOGGIO PARTENZA" )
      wire#w1
      Contact( "EV AV INDIETRO RIEMPITRICE" )
      Move(in := -90, out1 => "Blocco_dati_1"."pistone riempitore av ind x")
   END_RUNG
   RUNG wire#w1
      I_Contact( "EV AV INDIETRO RIEMPITRICE" )
      Move(in := 0, out1 => "Blocco_dati_1"."pistone riempitore av ind x")
   END_RUNG
   RUNG wire#w1
      Contact( "EV BECCUCCIO RIEMPITRICE" )
      Move(in := 30, out1 => "Blocco_dati_1"."riempitore su giu y")
   END_RUNG
   RUNG wire#w1
      I_Contact( "EV BECCUCCIO RIEMPITRICE" )
      Move(in := 0, out1 => "Blocco_dati_1"."riempitore su giu y")
   END_RUNG
   RUNG wire#w1
      Contact( "Blocco_dati_1"."FLACONE IN RIEMPIMENTO" )
      Contact( "EV BECCUCCIO RIEMPITRICE" )
      Contact( "EV RIEMPIMENTO FLACONE" )
      S_Coil( "Blocco_dati_1"."FLACONE PIENO" )
   END_RUNG
   RUNG wire#w1
      Contact( "Blocco_dati_1"."FLACONE PIENO" )
      Move(in := 1, out1 => "Blocco_dati_1"."riempimento flacone")
   END_RUNG
   RUNG wire#w1
      I_Contact( "Blocco_dati_1"."FLACONE PIENO" )
      Move(in := 0, out1 => "Blocco_dati_1"."riempimento flacone")
   END_RUNG
   // the same network as SCL:
   #_w1 := NOT "Blocco_dati_1"."APPOGGIO PARTENZA";
   IF #_w1 AND "EV AV INDIETRO RIEMPITRICE" THEN
       "Blocco_dati_1"."pistone riempitore av ind x" := -90;
   END_IF;
   IF #_w1 AND NOT "EV AV INDIETRO RIEMPITRICE" THEN
       "Blocco_dati_1"."pistone riempitore av ind x" := 0;
   END_IF;
   IF #_w1 AND "EV BECCUCCIO RIEMPITRICE" THEN "Blocco_dati_1"."riempitore su giu y" := 30; END_IF;
   IF #_w1 AND NOT "EV BECCUCCIO RIEMPITRICE" THEN "Blocco_dati_1"."riempitore su giu y" := 0; END_IF;
   IF #_w1 AND "Blocco_dati_1"."FLACONE IN RIEMPIMENTO" AND "EV BECCUCCIO RIEMPITRICE" AND "EV RIEMPIMENTO FLACONE" THEN
       "Blocco_dati_1"."FLACONE PIENO" := TRUE;
   END_IF;
   IF #_w1 AND "Blocco_dati_1"."FLACONE PIENO" THEN "Blocco_dati_1"."riempimento flacone" := 1; END_IF;
   IF #_w1 AND NOT "Blocco_dati_1"."FLACONE PIENO" THEN "Blocco_dati_1"."riempimento flacone" := 0; END_IF;
END_REGION

REGION Network 6: SENSORI PISTONE 1
   IF "EV PISTONE 1 MISURA" THEN
       "Blocco_dati_1"."SENSORE INDIETRO PISTONE_1" := 0;
       "Blocco_dati_1"."SENSORE AVANTI PISTONE_1" := 1;
   END_IF;
   "IEC_Timer_0_DB_3".TON(IN := "EV PISTONE 1 MISURA", PT := T#200MS);
   "FC PISTONE 1 AVANTI" := "IEC_Timer_0_DB_3".Q;
   #_w1 := NOT "EV PISTONE 1 MISURA";
   IF #_w1 THEN
       "Blocco_dati_1"."SENSORE AVANTI PISTONE_1" := 0;
       "Blocco_dati_1"."SENSORE INDIETRO PISTONE_1" := 1;
   END_IF;
   "IEC_Timer_0_DB_4".TON(IN := #_w1, PT := T#200MS);
   "FC PISTONE 1 INDIETRO" := "IEC_Timer_0_DB_4".Q;
END_REGION

REGION Network 7: SENSORI PISTONE 2
   IF "EV PISTONE 2 MISURA" THEN
       "Blocco_dati_1"."SENSORE INDIETRO PISTONE_2" := 0;
       "Blocco_dati_1"."SENSORE AVANTI PISTONE_2" := 1;
   END_IF;
   "IEC_Timer_0_DB_5".TON(IN := "EV PISTONE 2 MISURA", PT := T#200MS);
   "FC PISTONE 2 AVANTI" := "IEC_Timer_0_DB_5".Q;
   #_w1 := NOT "EV PISTONE 2 MISURA";
   IF #_w1 THEN
       "Blocco_dati_1"."SENSORE AVANTI PISTONE_2" := 0;
       "Blocco_dati_1"."SENSORE INDIETRO PISTONE_2" := 1;
   END_IF;
   "IEC_Timer_0_DB_6".TON(IN := #_w1, PT := T#200MS);
   "FC PISTONE 2 INDIETRO" := "IEC_Timer_0_DB_6".Q;
END_REGION

REGION Network 8: SENSORI PISTONE SU GIU
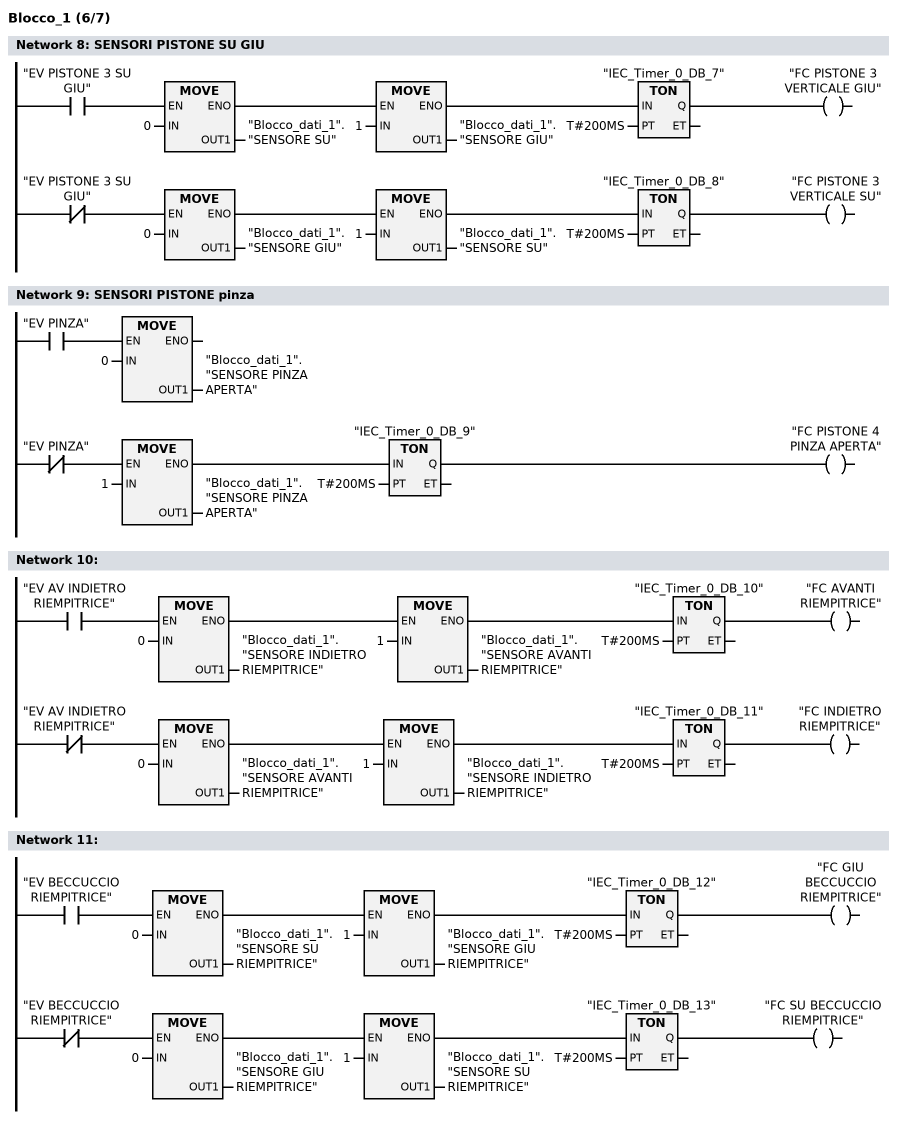
   IF "EV PISTONE 3 SU GIU" THEN
       "Blocco_dati_1"."SENSORE SU" := 0;
       "Blocco_dati_1"."SENSORE GIU" := 1;
   END_IF;
   "IEC_Timer_0_DB_7".TON(IN := "EV PISTONE 3 SU GIU", PT := T#200MS);
   "FC PISTONE 3 VERTICALE GIU" := "IEC_Timer_0_DB_7".Q;
   #_w1 := NOT "EV PISTONE 3 SU GIU";
   IF #_w1 THEN
       "Blocco_dati_1"."SENSORE GIU" := 0;
       "Blocco_dati_1"."SENSORE SU" := 1;
   END_IF;
   "IEC_Timer_0_DB_8".TON(IN := #_w1, PT := T#200MS);
   "FC PISTONE 3 VERTICALE SU" := "IEC_Timer_0_DB_8".Q;
END_REGION

REGION Network 9: SENSORI PISTONE pinza
   IF "EV PINZA" THEN "Blocco_dati_1"."SENSORE PINZA APERTA" := 0; END_IF;
   IF NOT "EV PINZA" THEN "Blocco_dati_1"."SENSORE PINZA APERTA" := 1; END_IF;
   "IEC_Timer_0_DB_9".TON(IN := NOT "EV PINZA", PT := T#200MS);
   "FC PISTONE 4 PINZA APERTA" := "IEC_Timer_0_DB_9".Q;
END_REGION

REGION Network 10
   IF "EV AV INDIETRO RIEMPITRICE" THEN
       "Blocco_dati_1"."SENSORE INDIETRO RIEMPITRICE" := 0;
       "Blocco_dati_1"."SENSORE AVANTI RIEMPITRICE" := 1;
   END_IF;
   "IEC_Timer_0_DB_10".TON(IN := "EV AV INDIETRO RIEMPITRICE", PT := T#200MS);
   "FC AVANTI RIEMPITRICE" := "IEC_Timer_0_DB_10".Q;
   #_w1 := NOT "EV AV INDIETRO RIEMPITRICE";
   IF #_w1 THEN
       "Blocco_dati_1"."SENSORE AVANTI RIEMPITRICE" := 0;
       "Blocco_dati_1"."SENSORE INDIETRO RIEMPITRICE" := 1;
   END_IF;
   "IEC_Timer_0_DB_11".TON(IN := #_w1, PT := T#200MS);
   "FC INDIETRO RIEMPITRICE" := "IEC_Timer_0_DB_11".Q;
END_REGION

REGION Network 11
   IF "EV BECCUCCIO RIEMPITRICE" THEN
       "Blocco_dati_1"."SENSORE SU RIEMPITRICE" := 0;
       "Blocco_dati_1"."SENSORE GIU RIEMPITRICE" := 1;
   END_IF;
   "IEC_Timer_0_DB_12".TON(IN := "EV BECCUCCIO RIEMPITRICE", PT := T#200MS);
   "FC GIU BECCUCCIO RIEMPITRICE" := "IEC_Timer_0_DB_12".Q;
   #_w1 := NOT "EV BECCUCCIO RIEMPITRICE";
   IF #_w1 THEN
       "Blocco_dati_1"."SENSORE GIU RIEMPITRICE" := 0;
       "Blocco_dati_1"."SENSORE SU RIEMPITRICE" := 1;
   END_IF;
   "IEC_Timer_0_DB_13".TON(IN := #_w1, PT := T#200MS);
   "FC SU BECCUCCIO RIEMPITRICE" := "IEC_Timer_0_DB_13".Q;
END_REGION

REGION Network 12: SENSORE PRESENZA PEZZO AL CARICO
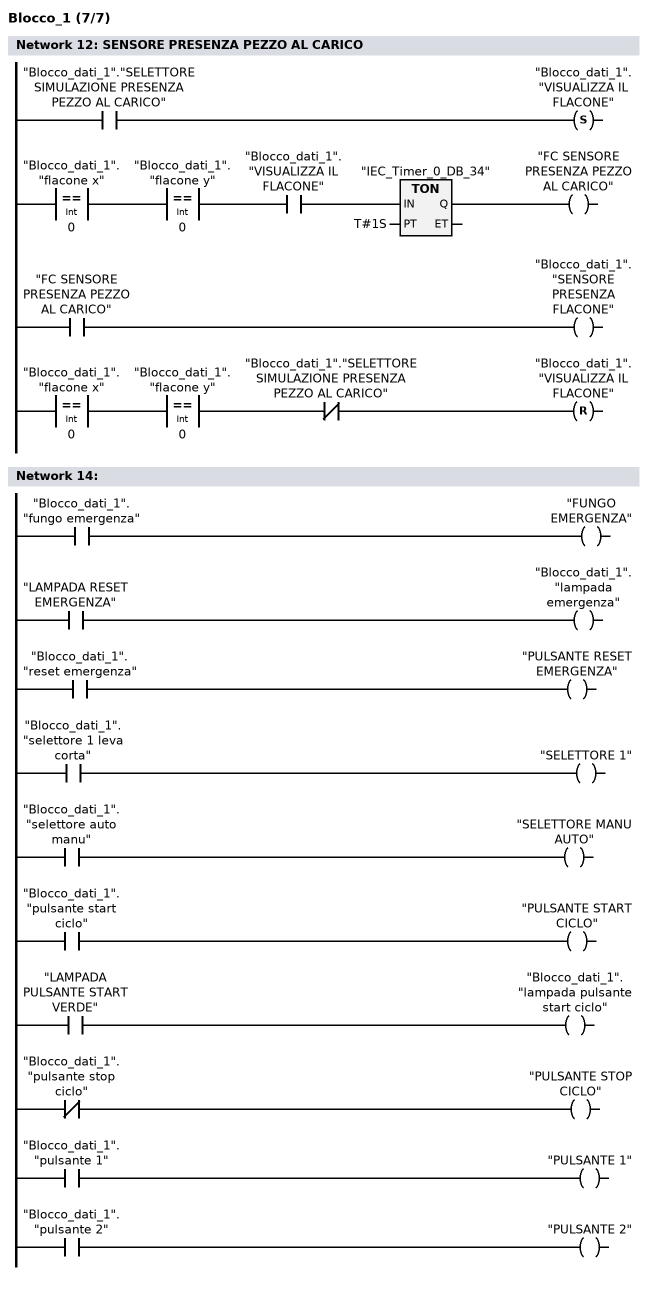
   IF "Blocco_dati_1"."SELETTORE SIMULAZIONE PRESENZA PEZZO AL CARICO" THEN
       "Blocco_dati_1"."VISUALIZZA IL FLACONE" := TRUE;
   END_IF;
   "IEC_Timer_0_DB_34".TON(IN := ("Blocco_dati_1"."flacone x" = 0) AND ("Blocco_dati_1"."flacone y" = 0) AND "Blocco_dati_1"."VISUALIZZA IL FLACONE",
                           PT := T#1S);
   "FC SENSORE PRESENZA PEZZO AL CARICO" := "IEC_Timer_0_DB_34".Q;
   "Blocco_dati_1"."SENSORE PRESENZA FLACONE" := "FC SENSORE PRESENZA PEZZO AL CARICO";
   IF ("Blocco_dati_1"."flacone x" = 0) AND ("Blocco_dati_1"."flacone y" = 0) AND NOT "Blocco_dati_1"."SELETTORE SIMULAZIONE PRESENZA PEZZO AL CARICO" THEN
       "Blocco_dati_1"."VISUALIZZA IL FLACONE" := FALSE;
   END_IF;
END_REGION

REGION Network 13: SENSORE PRESENZA PEZZO ALLO SCARICO
END_REGION

REGION Network 14
   RUNG wire#powerrail
      Contact( "Blocco_dati_1"."fungo emergenza" )
      Coil( "FUNGO EMERGENZA" )
   END_RUNG
   RUNG wire#powerrail
      Contact( "LAMPADA RESET EMERGENZA" )
      Coil( "Blocco_dati_1"."lampada emergenza" )
   END_RUNG
   RUNG wire#powerrail
      Contact( "Blocco_dati_1"."reset emergenza" )
      Coil( "PULSANTE RESET EMERGENZA" )
   END_RUNG
   RUNG wire#powerrail
      Contact( "Blocco_dati_1"."selettore 1 leva corta" )
      Coil( "SELETTORE 1" )
   END_RUNG
   RUNG wire#powerrail
      Contact( "Blocco_dati_1"."selettore auto manu" )
      Coil( "SELETTORE MANU  AUTO" )
   END_RUNG
   RUNG wire#powerrail
      Contact( "Blocco_dati_1"."pulsante start ciclo" )
      Coil( "PULSANTE START CICLO" )
   END_RUNG
   RUNG wire#powerrail
      Contact( "LAMPADA PULSANTE START VERDE" )
      Coil( "Blocco_dati_1"."lampada pulsante start ciclo" )
   END_RUNG
   RUNG wire#powerrail
      I_Contact( "Blocco_dati_1"."pulsante stop ciclo" )
      Coil( "PULSANTE STOP CICLO" )
   END_RUNG
   RUNG wire#powerrail
      Contact( "Blocco_dati_1"."pulsante 1" )
      Coil( "PULSANTE 1" )
   END_RUNG
   RUNG wire#powerrail
      Contact( "Blocco_dati_1"."pulsante 2" )
      Coil( "PULSANTE 2" )
   END_RUNG
   // the same network as SCL:
   "FUNGO EMERGENZA" := "Blocco_dati_1"."fungo emergenza";
   "Blocco_dati_1"."lampada emergenza" := "LAMPADA RESET EMERGENZA";
   "PULSANTE RESET EMERGENZA" := "Blocco_dati_1"."reset emergenza";
   "SELETTORE 1" := "Blocco_dati_1"."selettore 1 leva corta";
   "SELETTORE MANU  AUTO" := "Blocco_dati_1"."selettore auto manu";
   "PULSANTE START CICLO" := "Blocco_dati_1"."pulsante start ciclo";
   "Blocco_dati_1"."lampada pulsante start ciclo" := "LAMPADA PULSANTE START VERDE";
   "PULSANTE STOP CICLO" := NOT "Blocco_dati_1"."pulsante stop ciclo";
   "PULSANTE 1" := "Blocco_dati_1"."pulsante 1";
   "PULSANTE 2" := "Blocco_dati_1"."pulsante 2";
END_REGION
END_FUNCTION

(* ===== HMI "HMI_RT_1" =====
system functions are stored by id; their names below are inferred from use
connection "HMI_Collegamento_1": ETHERNET, SMART_S7_1200_OMS

HMI tags "Tabella delle variabili standard"
   "Blocco_dati_1_pistone 1  X" : Int = PLC Blocco_dati_1."pistone 1  X", 100 ms
   "Blocco_dati_1_pistone 2  X" : Int = PLC Blocco_dati_1."pistone 2  X", 100 ms
   "Blocco_dati_1_pistone 2 Y" : Int = PLC Blocco_dati_1."pistone 2 Y", 100 ms
   "Blocco_dati_1_pistone 3  X" : Int = PLC Blocco_dati_1."pistone 3  X", 100 ms
   "Blocco_dati_1_pistone 3 Y" : Int = PLC Blocco_dati_1."pistone 3 Y", 100 ms
   "Blocco_dati_1_corpo pinza x" : Int = PLC Blocco_dati_1."corpo pinza x", 100 ms
   "Blocco_dati_1_corpo pinza y" : Int = PLC Blocco_dati_1."corpo pinza y", 100 ms
   "Blocco_dati_1_dita aperte x" : Int = PLC Blocco_dati_1."dita aperte x", 100 ms
   "Blocco_dati_1_dita aperte y" : Int = PLC Blocco_dati_1."dita aperte y", 100 ms
   "Blocco_dati_1_dita chiuse x" : Int = PLC Blocco_dati_1."dita chiuse x", 100 ms
   "Blocco_dati_1_dita chiuse y" : Int = PLC Blocco_dati_1."dita chiuse y", 100 ms
   "Blocco_dati_1_pistone riempitore av ind x" : Int = PLC Blocco_dati_1."pistone riempitore av ind x", 100 ms
   "Blocco_dati_1_riempitore su giu" : Int = PLC Blocco_dati_1."riempitore su giu y", 100 ms
   "Blocco_dati_1_flacone x" : Int = PLC Blocco_dati_1."flacone x", 100 ms
   "Blocco_dati_1_flacone y" : Int = PLC Blocco_dati_1."flacone y", 100 ms
   "Blocco_dati_1_riempimento flacone" : Int = PLC Blocco_dati_1."riempimento flacone", 100 ms
   "Blocco_dati_1_pinza aperta" : Int = PLC Blocco_dati_1."pinza aperta", 100 ms
   "Blocco_dati_1_pinza chiusa" : Int = PLC Blocco_dati_1."pinza chiusa", 100 ms
   "Blocco_dati_1_lampada emergenza" : Bool = PLC Blocco_dati_1."lampada emergenza", 100 ms
   "Blocco_dati_1_reset emergenza" : Bool = PLC Blocco_dati_1."reset emergenza", 100 ms
   "Blocco_dati_1_pulsante start ciclo" : Bool = PLC Blocco_dati_1."pulsante start ciclo", 100 ms
   "Blocco_dati_1_pulsante stop ciclo" : Bool = PLC Blocco_dati_1."pulsante stop ciclo", 100 ms
   "Blocco_dati_1_pulsante 2" : Bool = PLC Blocco_dati_1."pulsante 2", 100 ms
   "Blocco_dati_1_pulsante 1" : Bool = PLC Blocco_dati_1."pulsante 1", 100 ms
   "Blocco_dati_1_selettore auto manu" : Bool = PLC Blocco_dati_1."selettore auto manu", 100 ms
   "Blocco_dati_1_MANUALI" : Byte = PLC Blocco_dati_1.MANUALI, 100 ms
   "Blocco_dati_1_pistone 1  Y" : Int = PLC Blocco_dati_1."pistone 1  Y", 100 ms
   "Blocco_dati_1_stelo pistone 2 x" : Int = PLC Blocco_dati_1."stelo pistone 2 x", 100 ms
   "Blocco_dati_1_stelo pistone 2 y" : Int = PLC Blocco_dati_1."stelo pistone 2 y", 100 ms
   "Blocco_dati_1_stelo pistone 3 x" : Int = PLC Blocco_dati_1."stelo pistone 3 x", 100 ms
   "Blocco_dati_1_stelo pistone 3 y" : Int = PLC Blocco_dati_1."stelo pistone 3 y", 100 ms
   "Blocco_dati_1_pistone riempitore av ind y" : Int = PLC Blocco_dati_1."pistone riempitore av ind y", 100 ms
   "Blocco_dati_1_SENSORE INDIETRO PISTONE_1" : Byte = PLC Blocco_dati_1."SENSORE INDIETRO PISTONE_1", 100 ms
   "Blocco_dati_1_SENSORE AVANTI PISTONE_1" : Byte = PLC Blocco_dati_1."SENSORE AVANTI PISTONE_1", 100 ms
   "Blocco_dati_1_SENSORE INDIETRO PISTONE_2" : Byte = PLC Blocco_dati_1."SENSORE INDIETRO PISTONE_2", 100 ms
   "Blocco_dati_1_SENSORE AVANTI PISTONE_2" : Byte = PLC Blocco_dati_1."SENSORE AVANTI PISTONE_2", 100 ms
   "Blocco_dati_1_SENSORE SU" : Byte = PLC Blocco_dati_1."SENSORE SU", 100 ms
   "Blocco_dati_1_SENSORE GIU" : Byte = PLC Blocco_dati_1."SENSORE GIU", 100 ms
   "Blocco_dati_1_SENSORE PINZA APERTA" : Byte = PLC Blocco_dati_1."SENSORE PINZA APERTA", 100 ms
   "Blocco_dati_1_SENSORE AVANTI RIEMPITRICE" : Byte = PLC Blocco_dati_1."SENSORE AVANTI RIEMPITRICE", 100 ms
   "Blocco_dati_1_SENSORE INDIETRO RIEMPITRICE" : Byte = PLC Blocco_dati_1."SENSORE INDIETRO RIEMPITRICE", 100 ms
   "Blocco_dati_1_SENSORE PRESENZA FLACONE" : Bool = PLC Blocco_dati_1."SENSORE PRESENZA FLACONE", 100 ms
   "Blocco_dati_1_SENSORE PRESENZA PEZZO ALLO SCARICO" : Byte = PLC Blocco_dati_1."RISPOSTA TELECAMERA DI ISPEZIONE", 100 ms
   "Blocco_dati_1_SENSORE SU RIEMPITRICE" : Byte = PLC Blocco_dati_1."SENSORE SU RIEMPITRICE", 100 ms
   "Blocco_dati_1_SENSORE GIU RIEMPITRICE" : Byte = PLC Blocco_dati_1."SENSORE GIU RIEMPITRICE", 100 ms
   "Blocco_dati_1_fungo emergenza" : Bool = PLC Blocco_dati_1."fungo emergenza", 100 ms
   "Blocco_dati_1_lampada pulsante start ciclo" : Bool = PLC Blocco_dati_1."lampada pulsante start ciclo", 100 ms
   "Blocco_dati_1_selettore 1 leva corta" : Bool = PLC Blocco_dati_1."selettore 1 leva corta", 100 ms
   "Blocco_dati_1_VISUALIZZA IL FLACONE" : Bool = PLC Blocco_dati_1."VISUALIZZA IL FLACONE", 1 s
   "Blocco_dati_1_SELETTORE SIMULAZIONE PRESENZA PEZZO AL CARICO" : Bool = PLC Blocco_dati_1."SELETTORE SIMULAZIONE PRESENZA PEZZO AL CARICO", 1 s
   "RISERVA 1" : Bool = PLC "RISERVA 1" AT %I0.6, 1 s
   "RISERVA 2" : Bool = PLC "RISERVA 2" AT %I0.7, 1 s
   "RISERVA 3" : Bool = PLC "RISERVA 3" AT %I8.2, 1 s

HMI tags "1_VariabiliPerManuale"
   "0-DB-Generale_6-VisibilitaComandiManuali" : Bool = PLC "0-DB-Generale".5-VisibilitaComandiManuali, 1 s
   "0-DB-Generale_6-PulsanteAvantiPistone1" : Bool = PLC "0-DB-Generale".6-PulsanteAvantiPistone1, 1 s
   "0-DB-Generale_6-PulsanteIndietroPistone1" : Bool = PLC "0-DB-Generale".6-PulsanteIndietroPistone1, 1 s
   "0-DB-Generale_6-PulsanteAvantiPistone2" : Bool = PLC "0-DB-Generale".6-PulsanteAvantiPistone2 AT %DB1.DBX0.0, 1 s
   "0-DB-Generale_6-PulsanteIndietroPistone2" : Bool = PLC "0-DB-Generale".6-PulsanteIndietroPistone2 AT %DB1.DBX0.0, 1 s
   "0-DB-Generale_6-PulsanteGiuPistone3" : Bool = PLC "0-DB-Generale".6-PulsanteGiuPistone3 AT %DB1.DBX0.0, 1 s
   "0-DB-Generale_6-PulsanteSuPistone3" : Bool = PLC "0-DB-Generale".6-PulsanteSuPistone3 AT %DB1.DBX0.0, 1 s
   "0-DB-Generale_6-PulsanteChiudiPinza" : Bool = PLC "0-DB-Generale".6-PulsanteChiudiPinza AT %DB1.DBX0.0, 1 s
   "0-DB-Generale_6-PulsanteApriPinza" : Bool = PLC "0-DB-Generale".6-PulsanteApriPinza AT %DB1.DBX0.0, 1 s
   "0-DB-Generale_6-PulsanteAvantiPistone5Riempitrice" : Bool = PLC "0-DB-Generale".6-PulsanteAvantiPistone5Riempitrice AT %DB1.DBX0.0, 1 s
   "0-DB-Generale_6-PulsanteIndietroPistone5Riempitrice" : Bool = PLC "0-DB-Generale".6-PulsanteIndietroPistone5Riempitrice AT %DB1.DBX0.0, 1 s
   "0-DB-Generale_6-PulsanteGiuPistone6Beccuccio" : Bool = PLC "0-DB-Generale".6-PulsanteGiuPistone6Beccuccio AT %DB1.DBX0.0, 1 s
   "0-DB-Generale_6-PulsanteSuPistone6Beccuccio" : Bool = PLC "0-DB-Generale".6-PulsanteSuPistone6Beccuccio AT %DB1.DBX0.0, 1 s
   "0-DB-Generale_6-PulsanteRiempimento" : Bool = PLC "0-DB-Generale".6-PulsanteRiempimento AT %DB1.DBX0.0, 1 s

HMI tags "2_VariabiliHmiUtilities"
   "0-DB-Generale_5-HMI => Current time of day" : DTL = PLC "0-DB-Generale"."5-HMI => Current time of day", 1 s
   "0-DB-Generale_0-StatoMacchina" : Int = PLC "0-DB-Generale".0-StatoMacchina AT %DB1.DBX0.0, 1 s
   "0-DB-Generale_5-HMI => Only current time" : Time_Of_Day = PLC "0-DB-Generale"."5-HMI => Only current time", 1 s
   "0-DB-Generale_5-HMI => Only current date" : Date = PLC "0-DB-Generale"."5-HMI => Only current date", 1 s
   "0-DB-Generale_5-HMI => Timer ultima eccezione" : Bool = PLC "0-DB-Generale"."5-HMI => Timer ultima eccezione", 1 s

HMI tags "3_DatiPlc"
   "0-DB-Generale_0-IdCommessa" : Int = PLC "0-DB-Generale".0-IdCommessa, 1 s
   "0-DB-Generale_0-IdMacchinario" : Int = PLC "0-DB-Generale".0-IdMacchinario, 1 s
   "0-DB-Generale_0-IdProdotto" : Int = PLC "0-DB-Generale".0-IdProdotto, 1 s
   "0-DB-Generale_0-PezziTotali" : Int = PLC "0-DB-Generale".0-PezziTotali, 1 s
   "0-DB-Generale_0-TimeStampAttuale" : DTL = PLC "0-DB-Generale".0-TimeStampAttuale, 1 s
   "0-DB-Generale_0-PezziBuoniProdotti" : Int = PLC "0-DB-Generale".0-PezziBuoniProdotti, 1 s
   "0-DB-Generale_0-PezziScartiProdotti" : Int = PLC "0-DB-Generale".0-PezziScartiProdotti, 1 s
   "0-DB-Generale_0-MinutiDiLavoro" : Int = PLC "0-DB-Generale".0-MinutiDiLavoro, 1 s
   "0-DB-Generale_0-TImeStampInizioCiclo" : Int = PLC "0-DB-Generale".0-TImeStampInizioCiclo, 1 s
   "0-DB-Generale_0-TimeStampFineCiclo" : Int = PLC "0-DB-Generale".0-TimeStampFineCiclo, 1 s
   "0-DB-Generale_0-IdAttuatori" : Array [0..1] of Int = PLC "0-DB-Generale".0-IdAttuatori, 1 s
   "0-DB-Generale_0-NumeroAttivazioniAttuatori" : Array [0..1] of Int = PLC "0-DB-Generale".0-NumeroAttivazioniAttuatori, 1 s
   "0-DB-Generale_0-IdSensori" : Array [0..1] of Int = PLC "0-DB-Generale".0-IdSensori, 1 s
   "0-DB-Generale_0-NumeroAttivazioniSensori" : Array [0..1] of Int = PLC "0-DB-Generale".0-NumeroAttivazioniSensori, 1 s
   "0-DB-Generale_0-PezziPerMinuto" : Real = PLC "0-DB-Generale".0-PezziPerMinuto, 1 s
   "0-DB-Generale_0-Allarmi" : Array [0..1] of Bool = PLC "0-DB-Generale".0-Allarmi, 1 s

text list "Elenco_testi_1": 0 ''; 1 'AP CH PINZA'; 2 'SU GIU PINZA'; 3 'AV INDIETRO PISTONE 1'; 4 'AV INDIETRO PISTONE 2'; 5 'AV IND RIEMPITRICE'; 6 'SI GIU BECCUCCIO'

screen "1_principale" 800x480
   Rectangle "Rettangolo_23" at 644,269 size 7x55
      DirectMovement <- "Blocco_dati_1_pistone riempitore av ind x"
      DirectMovement <- "Blocco_dati_1_riempitore su giu"
   Rectangle "Rettangolo_4" at 309,39 size 17x165
      DirectMovement <- "Blocco_dati_1_stelo pistone 3 x"
      DirectMovement <- "Blocco_dati_1_stelo pistone 3 y"
   Rectangle "Rettangolo_2" at 78,149 size 222x17
      DirectMovement <- "Blocco_dati_1_stelo pistone 2 x"
      DirectMovement <- "Blocco_dati_1_stelo pistone 2 y"
   Rectangle "Rettangolo_1" at 50,141 size 225x35
      DirectMovement <- "Blocco_dati_1_pistone 2  X"
      DirectMovement <- "Blocco_dati_1_pistone 2 Y"
   Rectangle "Rettangolo_3" at 300,11 size 35x173
      DirectMovement <- "Blocco_dati_1_pistone 3  X"
      DirectMovement <- "Blocco_dati_1_pistone 3 Y"
   Rectangle "Rettangolo_5" at 280,205 size 75x20
      DirectMovement <- "Blocco_dati_1_corpo pinza x"
      DirectMovement <- "Blocco_dati_1_corpo pinza y"
   Rectangle "Rettangolo_6" at 280,225 size 16x37
      Visibility <- "Blocco_dati_1_pinza aperta"
      DirectMovement <- "Blocco_dati_1_dita aperte x"
      DirectMovement <- "Blocco_dati_1_dita aperte y"
   Rectangle "Rettangolo_7" at 339,225 size 16x37
      Visibility <- "Blocco_dati_1_pinza aperta"
      DirectMovement <- "Blocco_dati_1_dita aperte x"
      DirectMovement <- "Blocco_dati_1_dita aperte y"
   Rectangle "Rettangolo_8" at 309,333 size 18x49
      DirectMovement <- "Blocco_dati_1_flacone x"
      DirectMovement <- "Blocco_dati_1_flacone y"
      Appearance <- "Blocco_dati_1_riempimento flacone"
      Visibility <- "Blocco_dati_1_VISUALIZZA IL FLACONE"
   Rectangle "Rettangolo_9" at 328,225 size 16x37
      Visibility <- "Blocco_dati_1_pinza chiusa"
      DirectMovement <- "Blocco_dati_1_dita chiuse y"
      DirectMovement <- "Blocco_dati_1_dita chiuse x"
   Rectangle "Rettangolo_10" at 293,225 size 16x37
      Visibility <- "Blocco_dati_1_pinza chiusa"
      DirectMovement <- "Blocco_dati_1_dita chiuse y"
      DirectMovement <- "Blocco_dati_1_dita chiuse x"
   Rectangle "Rettangolo_11" at 50,92 size 160x48
      DirectMovement <- "Blocco_dati_1_pistone 1  X"
      DirectMovement <- "Blocco_dati_1_pistone 1  Y"
   Circle "Cerchio_1" at 68,96 size 10x10
      DirectMovement <- "Blocco_dati_1_pistone 1  X"
      DirectMovement <- "Blocco_dati_1_pistone 1  Y"
      Visibility <- "Blocco_dati_1_SENSORE INDIETRO PISTONE_1"
   Circle "Cerchio_3" at 197,96 size 10x10
      DirectMovement <- "Blocco_dati_1_pistone 1  X"
      DirectMovement <- "Blocco_dati_1_pistone 1  Y"
      Visibility <- "Blocco_dati_1_SENSORE AVANTI PISTONE_1"
   Circle "Cerchio_2" at 67,148 size 10x10
      DirectMovement <- "Blocco_dati_1_pistone 2  X"
      DirectMovement <- "Blocco_dati_1_pistone 2 Y"
      Visibility <- "Blocco_dati_1_SENSORE INDIETRO PISTONE_2"
   Circle "Cerchio_4" at 255,148 size 10x10
      DirectMovement <- "Blocco_dati_1_pistone 2  X"
      DirectMovement <- "Blocco_dati_1_pistone 2 Y"
      Visibility <- "Blocco_dati_1_SENSORE AVANTI PISTONE_2"
   Circle "Cerchio_5" at 316,170 size 10x10
      DirectMovement <- "Blocco_dati_1_pistone 3  X"
      DirectMovement <- "Blocco_dati_1_pistone 3 Y"
      Visibility <- "Blocco_dati_1_SENSORE GIU"
   Circle "Cerchio_6" at 316,16 size 10x10
      DirectMovement <- "Blocco_dati_1_pistone 3  X"
      DirectMovement <- "Blocco_dati_1_pistone 3 Y"
      Visibility <- "Blocco_dati_1_SENSORE SU"
   Circle "Cerchio_7" at 343,209 size 10x10
      DirectMovement <- "Blocco_dati_1_corpo pinza x"
      DirectMovement <- "Blocco_dati_1_corpo pinza y"
      Visibility <- "Blocco_dati_1_SENSORE PINZA APERTA"
   Rectangle "Rettangolo_19" at 674,286 size 116x21
      DirectMovement <- "Blocco_dati_1_pistone riempitore av ind x"
      DirectMovement <- "Blocco_dati_1_pistone riempitore av ind y"
   Circle "Cerchio_10" at 704,307 size 10x10
      Visibility <- "Blocco_dati_1_SENSORE AVANTI RIEMPITRICE"
   Circle "Cerchio_11" at 777,308 size 10x10
      Visibility <- "Blocco_dati_1_SENSORE INDIETRO RIEMPITRICE"
   Rectangle "Rettangolo_21" at 620,268 size 57x52
      DirectMovement <- "Blocco_dati_1_pistone riempitore av ind x"
      DirectMovement <- "Blocco_dati_1_pistone riempitore av ind y"
   TextField "Casella di testo_1" at 733,1 size 47x18; Text 'Fungo'
   TextField "Casella di testo_2" at 720,13 size 71x18; Text 'Emergenza'
   Button "Pulsante_2" at 740,120 size 40x41; TextOff 'Text'
      Appearance <- "Blocco_dati_1_lampada emergenza"
      on Press: function_b14e0dd5("Blocco_dati_1_reset emergenza", 0)
   TextField "Casella di testo_3" at 739,92 size 40x18; Text 'Reset'
   TextField "Casella di testo_4" at 726,103 size 71x18; Text 'Emergenza'
   Button "Pulsante_1" at 673,120 size 40x41; TextOff 'Text'
      on Press: function_b14e0dd5("Blocco_dati_1_pulsante stop ciclo", 0)
   TextField "Casella di testo_5" at 672,92 size 35x18; Text 'Stop'
   TextField "Casella di testo_6" at 659,103 size 47x18; Text 'ciclo'
   Button "Pulsante_3" at 623,120 size 40x41; TextOff 'Text'
      on Press: function_b14e0dd5("Blocco_dati_1_pulsante start ciclo", 0)
      Appearance <- "Blocco_dati_1_lampada pulsante start ciclo"
   TextField "Casella di testo_7" at 623,92 size 41x18; Text 'Start'
   TextField "Casella di testo_8" at 624,103 size 33x18; Text 'Ciclo'
   Switch "Interruttore_1" at 738,188 size 41x39; CaptionText 'Switch'; TextOff 'OFF'; TextOn 'ON'; PictureOff "SELETTORE PER SIEMENS SX"; PictureOn "SELETTORE PER SIEMENS DX"
      ProcessValue <- "Blocco_dati_1_selettore auto manu"
   Button "Pulsante_4" at 671,39 size 40x41; TextOff 'Text'
      on Press: function_b14e0dd5("Blocco_dati_1_pulsante 2", 0)
   TextField "Casella di testo_9" at 665,17 size 48x18; Text 'PULS 2'
   Button "Pulsante_5" at 622,39 size 40x41; TextOff 'Text'
      on Press: function_b14e0dd5("Blocco_dati_1_pulsante 1", 0)
   TextField "Casella di testo_10" at 616,17 size 48x18; Text 'PULS 1'
   TextField "Casella di testo_11" at 724,166 size 70x18; Text 'MAN AUTO'
   SymbolicIOField "Campo I/O simbolico_1" at 604,232 size 194x30; TextOff '0'; TextOn '1'; TextList "Elenco_testi_1"
      ProcessValue <- "Blocco_dati_1_MANUALI"
   Rectangle "Rettangolo_27" at 331,364 size 9x15
      Appearance <- "Blocco_dati_1_SENSORE PRESENZA FLACONE"
   Rectangle "Rettangolo_29" at 446,353 size 17x28
      Appearance <- "Blocco_dati_1_SENSORE PRESENZA PEZZO ALLO SCARICO"
   Circle "Cerchio_13" at 644,274 size 10x10
      Visibility <- "Blocco_dati_1_SENSORE SU RIEMPITRICE"
      DirectMovement <- "Blocco_dati_1_pistone riempitore av ind x"
      DirectMovement <- "Blocco_dati_1_pistone riempitore av ind y"
   Circle "Cerchio_14" at 644,303 size 10x10
      Visibility <- "Blocco_dati_1_SENSORE GIU RIEMPITRICE"
      DirectMovement <- "Blocco_dati_1_pistone riempitore av ind x"
      DirectMovement <- "Blocco_dati_1_pistone riempitore av ind y"
   TextField "Casella di testo_12" at 124,107 size 13x20; Text '1'
      DirectMovement <- "Blocco_dati_1_pistone 1  X"
      DirectMovement <- "Blocco_dati_1_pistone 1  Y"
   TextField "Casella di testo_13" at 144,149 size 13x20; Text '2'
      DirectMovement <- "Blocco_dati_1_pistone 2  X"
      DirectMovement <- "Blocco_dati_1_pistone 2 Y"
   TextField "Casella di testo_14" at 311,80 size 13x20; Text '3'
      DirectMovement <- "Blocco_dati_1_pistone 3  X"
      DirectMovement <- "Blocco_dati_1_pistone 3 Y"
   TextField "Casella di testo_15" at 310,205 size 13x20; Text '4'
      DirectMovement <- "Blocco_dati_1_corpo pinza x"
      DirectMovement <- "Blocco_dati_1_corpo pinza y"
   TextField "Casella di testo_16" at 738,288 size 13x20; Text '5'
   Switch "Interruttore_3" at 644,188 size 41x39; CaptionText 'Switch'; TextOff 'OFF'; TextOn 'ON'; PictureOff "SELETTORE PER SIEMENS SX"; PictureOn "SELETTORE PER SIEMENS DX"
      ProcessValue <- "Blocco_dati_1_selettore 1 leva corta"
   TextField "Casella di testo_17" at 635,179 size 53x18; Text '0 1'
   TextField "Casella di testo_18" at 623,166 size 85x18; Text 'SELETTORE 1'
   Switch "Interruttore_4" at 302,435 size 41x39; CaptionText 'Switch'; TextOff 'OFF'; TextOn 'ON'; PictureOff "SELETTORE PER SIEMENS SX"; PictureOn "SELETTORE PER SIEMENS DX"
      ProcessValue <- "Blocco_dati_1_SELETTORE SIMULAZIONE PRESENZA PEZZO AL CARICO"
   TextField "Casella di testo_19" at 293,425 size 53x18; Text '0 1'
   TextField "Casella di testo_20" at 107,442 size 182x18; Text 'PRESENZA PEZZO AL CARICO'
   Switch "Interruttore_5" at 60,32 size 41x39; CaptionText 'Switch'; TextOff 'OFF'; TextOn 'ON'; PictureOff "SELETTORE PER SIEMENS SX"; PictureOn "SELETTORE PER SIEMENS DX"
      ProcessValue <- "RISERVA 1"
   TextField "Casella di testo_21" at 51,23 size 53x18; Text '0 1'
   TextField "Casella di testo_22" at 45,10 size 67x18; Text 'SCORTA 1'
   Switch "Interruttore_6" at 142,34 size 41x39; CaptionText 'Switch'; TextOff 'OFF'; TextOn 'ON'; PictureOff "SELETTORE PER SIEMENS SX"; PictureOn "SELETTORE PER SIEMENS DX"
      ProcessValue <- "RISERVA 2"
   TextField "Casella di testo_23" at 133,25 size 53x18; Text '0 1'
   TextField "Casella di testo_24" at 124,11 size 67x18; Text 'SCORTA 2'
   Switch "Interruttore_7" at 227,34 size 41x39; CaptionText 'Switch'; TextOff 'OFF'; TextOn 'ON'; PictureOff "SELETTORE PER SIEMENS SX"; PictureOn "SELETTORE PER SIEMENS DX"
      ProcessValue <- "RISERVA 3"
   TextField "Casella di testo_25" at 218,25 size 53x18; Text '0 1'
   TextField "Casella di testo_26" at 210,12 size 67x18; Text 'SCORTA 3'
   Switch "Interruttore_8" at 740,45 size 37x34; CaptionText 'Switch'; TextOff 'OFF'; TextOn 'ON'; PictureOn "fungo per siemens 2_2"; PictureOff "fungo per siemens 1_2"
      ProcessValue <- "Blocco_dati_1_fungo emergenza"
   Softkey "Softkey_F1" at 0,0 size 0x0
      on KeyDown: ActivateScreen("1_principale", 0)
   Softkey "Softkey_F2" at 0,0 size 0x0
      on KeyDown: ActivateScreen("2_HomeBeforeLogin", 0)
   Softkey "Softkey_F3" at 0,0 size 0x0
      on KeyDown: ActivateScreen("3_HomeAfterLogin", 0)
   Softkey "Softkey_F4" at 0,0 size 0x0
      on KeyDown: ActivateScreen("4_Manuali", 0)

screen "3_HomeAfterLogin" 800x480
   Button "Button_2" at 0,408 size 130x71; TextOff 'Pag 1'
   Button "Button_3" at 130,408 size 130x71; TextOff 'Manuali'
      on Click: ActivateScreen("4_Manuali", 0)
   Button "Button_4" at 260,408 size 130x71; TextOff 'Pag 3'
   Button "Button_5" at 390,408 size 130x71; TextOff 'Pag 4'
   Button "Button_6" at 520,408 size 130x71; TextOff 'Pag 5'
   Button "Button_7" at 650,408 size 130x71; TextOff 'Pag 6'
   IOField "I/O field_1" at 139,17 size 121x32; FormatPattern 99
      ProcessValue <- "0-DB-Generale_5-HMI => Only current date"
   IOField "I/O field_2" at 151,41 size 96x32; FormatPattern 99999999999999999999
      ProcessValue <- "0-DB-Generale_5-HMI => Only current time"
   Circle "Circle_1" at 327,10 size 63x63
      Appearance <- "0-DB-Generale_0-StatoMacchina"
   TextField "start" at 397,0 size 55x28; Text 'Start'
      Visibility <- "0-DB-Generale_0-StatoMacchina"
   TextField "campoTestoStop" at 397,56 size 51x28; Text 'Stop'
      Visibility <- "0-DB-Generale_0-StatoMacchina"
   TextField "campoTestoPronto" at 397,28 size 69x28; Text 'Ready'
      Visibility <- "0-DB-Generale_0-StatoMacchina"

screen "2_HomeBeforeLogin" 800x480
   Button "Button_1" at 710,15 size 84x53; TextOff 'login'; Authorization "Gestione utenti"
      on Click: ActivateScreen("3_HomeAfterLogin", 0)
   Button "Button_2" at 0,408 size 130x71; TextOff 'Pag 1'
      on Click: SetBit("0-DB-Generale_5-HMI => Timer ultima eccezione")
   Button "Button_3" at 130,408 size 130x71; TextOff 'Manuali'
      on Click: SetBit("0-DB-Generale_5-HMI => Timer ultima eccezione")
   Button "Button_4" at 260,408 size 130x71; TextOff 'Pag 3'
      on Click: SetBit("0-DB-Generale_5-HMI => Timer ultima eccezione")
   Button "Button_5" at 390,408 size 130x71; TextOff 'Pag 4'
      on Click: SetBit("0-DB-Generale_5-HMI => Timer ultima eccezione")
   Button "Button_6" at 520,408 size 130x71; TextOff 'Pag 5'
      on Click: SetBit("0-DB-Generale_5-HMI => Timer ultima eccezione")
   Button "Button_7" at 650,408 size 130x71; TextOff 'Pag 6'
      on Click: SetBit("0-DB-Generale_5-HMI => Timer ultima eccezione")
   Ellipse "Ellipse_1" at 628,81 size 148x66
      Visibility <- "0-DB-Generale_5-HMI => Timer ultima eccezione"
   TextField "Text field_4" at 647,104 size 116x20; Text 'Please log in first'
      Visibility <- "0-DB-Generale_5-HMI => Timer ultima eccezione"
   IOField "I/O field_1" at 139,17 size 121x32; FormatPattern 99
      ProcessValue <- "0-DB-Generale_5-HMI => Only current date"
   IOField "I/O field_2" at 151,41 size 96x32; FormatPattern 99999999999999999999
      ProcessValue <- "0-DB-Generale_5-HMI => Only current time"
   Circle "Circle_1" at 327,10 size 63x63
      Appearance <- "0-DB-Generale_0-StatoMacchina"
   TextField "start" at 397,0 size 55x28; Text 'Start'
      Visibility <- "0-DB-Generale_0-StatoMacchina"
   TextField "campoTestoStop" at 397,56 size 51x28; Text 'Stop'
      Visibility <- "0-DB-Generale_0-StatoMacchina"
   TextField "campoTestoPronto" at 397,28 size 69x28; Text 'Ready'
      Visibility <- "0-DB-Generale_0-StatoMacchina"

screen "4_Manuali" 800x480
   Circle "Circle_1" at 327,10 size 63x63
      Appearance <- "0-DB-Generale_0-StatoMacchina"
   TextField "start" at 397,0 size 55x28; Text 'Start'
      Visibility <- "0-DB-Generale_0-StatoMacchina"
   TextField "campoTestoStop" at 397,56 size 51x28; Text 'Stop'
      Visibility <- "0-DB-Generale_0-StatoMacchina"
   TextField "campoTestoPronto" at 397,28 size 69x28; Text 'Ready'
      Visibility <- "0-DB-Generale_0-StatoMacchina"
   Button "pulsantePagina1" at 0,408 size 130x71; TextOff 'Pag 1'
   Button "pulsantePaginaManuali" at 130,408 size 130x71; TextOff 'Manuali'
      on Click: ActivateScreen("4_Manuali", 0)
   Button "pulsantePagina3" at 260,408 size 130x71; TextOff 'Pag 3'
   Button "pulsantePagina4" at 390,408 size 130x71; TextOff 'Pag 4'
   Button "pulsantePagina5" at 520,408 size 130x71; TextOff 'Pag 5'
   Button "pulsantePagina6" at 650,408 size 130x71; TextOff 'Pag 6'
   IOField "campoIoData" at 139,17 size 121x32; FormatPattern 99999999999999999999
      ProcessValue <- "0-DB-Generale_5-HMI => Only current date"
   IOField "campoIoOra" at 151,41 size 96x32; FormatPattern 99999999999999999999
      ProcessValue <- "0-DB-Generale_5-HMI => Only current time"
   GraphicView "immagineManipolatore" at 72,84 size 331x300; Picture "vectorpaint"
      Visibility <- "0-DB-Generale_6-VisibilitaComandiManuali"
   GraphicView "immagineRiempitrice" at 520,172 size 249x189; Picture "iniettore_project_icon"
      Visibility <- "0-DB-Generale_6-VisibilitaComandiManuali"
   Button "pulsantePistone1Avanti" at 196,204 size 32x27; TextOff '➪'; PictureOff "Right_Arrow"
      Visibility <- "0-DB-Generale_6-VisibilitaComandiManuali"
      on Press: SetBit("0-DB-Generale_6-PulsanteAvantiPistone1")
      on Release: ResetBit("0-DB-Generale_6-PulsanteAvantiPistone1")
   Button "pulsantePistone1Indietro" at 151,204 size 32x27; TextOff 'Text'; PictureOff "Left_Arrow"
      Visibility <- "0-DB-Generale_6-VisibilitaComandiManuali"
      on Press: SetBit("0-DB-Generale_6-PulsanteIndietroPistone1")
      on Release: ResetBit("0-DB-Generale_6-PulsanteIndietroPistone1")
   Button "pulsantePistone2Indietro" at 151,236 size 32x27; TextOff '<'; PictureOff "Left_Arrow"
      Visibility <- "0-DB-Generale_6-VisibilitaComandiManuali"
      on Press: SetBit("0-DB-Generale_6-PulsanteIndietroPistone2")
      on Release: ResetBit("0-DB-Generale_6-PulsanteIndietroPistone2")
   Button "pulsantePistone2Avanti" at 240,236 size 32x27; TextOff '➪'; PictureOff "Right_Arrow"
      Visibility <- "0-DB-Generale_6-VisibilitaComandiManuali"
      on Press: SetBit("0-DB-Generale_6-PulsanteAvantiPistone2")
      on Release: ResetBit("0-DB-Generale_6-PulsanteAvantiPistone2")
   Button "pulsantePistone3Su" at 298,134 size 26x32; TextOff '<'; PictureOff "Up_Arrow"
      Visibility <- "0-DB-Generale_6-VisibilitaComandiManuali"
      on Press: SetBit("0-DB-Generale_6-PulsanteSuPistone3")
      on Release: ResetBit("0-DB-Generale_6-PulsanteSuPistone3")
   Button "pulsantePistone3Giu" at 298,233 size 26x32; TextOff '<'; PictureOff "Down_Arrow"
      Visibility <- "0-DB-Generale_6-VisibilitaComandiManuali"
      on Press: SetBit("0-DB-Generale_6-PulsanteGiuPistone3")
      on Release: ResetBit("0-DB-Generale_6-PulsanteGiuPistone3")
   Button "pulsanteChiudiPinza" at 324,302 size 36x32; TextOff '<'; PictureOff "image(1)"
      Visibility <- "0-DB-Generale_6-VisibilitaComandiManuali"
      on Press: SetBit("0-DB-Generale_6-PulsanteChiudiPinza")
      on Release: ResetBit("0-DB-Generale_6-PulsanteChiudiPinza")
   Button "pulsanteApriPinza" at 258,302 size 40x32; TextOff '<'; PictureOff "image"
      Visibility <- "0-DB-Generale_6-VisibilitaComandiManuali"
      on Press: SetBit("0-DB-Generale_6-PulsanteApriPinza")
      on Release: ResetBit("0-DB-Generale_6-PulsanteApriPinza")
   Button "pulsanteBeccuccioAvanti" at 502,203 size 32x27; TextOff 'Text'; PictureOff "Left_Arrow"
      Visibility <- "0-DB-Generale_6-VisibilitaComandiManuali"
      on Press: SetBit("0-DB-Generale_6-PulsanteAvantiPistone5Riempitrice")
      on Release: ResetBit("0-DB-Generale_6-PulsanteAvantiPistone5Riempitrice")
   Button "pulsanteBeccuccioIndietro" at 572,203 size 32x27; TextOff '➪'; PictureOff "Right_Arrow"
      Visibility <- "0-DB-Generale_6-VisibilitaComandiManuali"
      on Press: SetBit("0-DB-Generale_6-PulsanteIndietroPistone5Riempitrice")
      on Release: ResetBit("0-DB-Generale_6-PulsanteIndietroPistone5Riempitrice")
   Button "pulsanteBeccuccioGiu" at 563,275 size 21x28; TextOff '➪'; PictureOff "Down_Arrow"
      Visibility <- "0-DB-Generale_6-VisibilitaComandiManuali"
      on Press: SetBit("0-DB-Generale_6-PulsanteGiuPistone6Beccuccio")
      on Release: ResetBit("0-DB-Generale_6-PulsanteGiuPistone6Beccuccio")
   Button "pulsanteBeccuccioSu" at 563,247 size 21x28; TextOff '➪'; PictureOff "Up_Arrow"
      Visibility <- "0-DB-Generale_6-VisibilitaComandiManuali"
      on Press: SetBit("0-DB-Generale_6-PulsanteSuPistone6Beccuccio")
      on Release: ResetBit("0-DB-Generale_6-PulsanteSuPistone6Beccuccio")
   Button "pulsanteEstrudi" at 496,323 size 105x49; TextOff 'Riempimento'; PictureOff "Right_Arrow"
      Visibility <- "0-DB-Generale_6-VisibilitaComandiManuali"
      on Press: SetBit("0-DB-Generale_6-PulsanteRiempimento")
      on Release: ResetBit("0-DB-Generale_6-PulsanteRiempimento")
   Switch "selettoreRiempitriceManipolatore" at 566,99 size 175x32; CaptionText 'Switch'; TextOff 'Riempitrice'; TextOn 'Manipolatore'
      on SwitchOn: SetBit("0-DB-Generale_6-VisibilitaComandiManuali")
      on SwitchOff: ResetBit("0-DB-Generale_6-VisibilitaComandiManuali")
      ProcessValue <- "0-DB-Generale_6-VisibilitaComandiManuali"

screen "5_Dati" 800x480
   IOField "campoIoPezziBuoni" at 197,32 size 96x32; FormatPattern s99999
      ProcessValue <- "0-DB-Generale_0-PezziBuoniProdotti"
   IOField "campoIoPezziScarti" at 319,32 size 96x32; FormatPattern s99999
      ProcessValue <- "0-DB-Generale_0-PezziScartiProdotti"
   TextField "campoTestoPezziScarti" at 321,7 size 80x20; Text 'Pezzi Scarti'
   TextField "campoTestoPezziBuoni" at 197,7 size 77x20; Text 'Pezzi Buoni'
   IOField "campoIoTimestampInizio" at 22,159 size 96x32; FormatPattern s99999
      ProcessValue <- "0-DB-Generale_0-TImeStampInizioCiclo"
   TextField "campoTestoTimestampInizio" at 22,134 size 113x20; Text 'TimeStamp Inizio'
   IOField "campoIoTimestampFine" at 321,159 size 96x32; FormatPattern s99999
      ProcessValue <- "0-DB-Generale_0-TimeStampFineCiclo"
   TextField "campoTestoTimestampFine" at 321,134 size 104x20; Text 'TimeStamp Fine'
   IOField "campoIoPezziTotali" at 22,32 size 96x32; FormatPattern s99999
      ProcessValue <- "0-DB-Generale_0-PezziTotali"
   TextField "campoTestoPezziTotali" at 22,7 size 77x20; Text 'Pezzi Totali'
   IOField "campoIoMinutiDiLavoro" at 22,329 size 96x32; FormatPattern s99999
      ProcessValue <- "0-DB-Generale_0-MinutiDiLavoro"
   TextField "campoTestoMinutiDiLavoro" at 22,304 size 109x20; Text 'Minuti Di Lavoro'
   IOField "campoIoTimestampAttuale" at 197,226 size 96x32; FormatPattern s99999
      ProcessValue <- "0-DB-Generale_0-TimeStampFineCiclo"
   TextField "campoTestoTimestampAttuale" at 197,205 size 464x20; Text 'TimeStamp Attuale (legato a Timestamp fine, dtl tipo non supportato?)'
   IOField "campoIoPezziAlMinuto" at 443,32 size 96x32; FormatPattern s999999999.999
      ProcessValue <- "0-DB-Generale_0-PezziPerMinuto"
   TextField "campoTestoPezziAlMinuto" at 443,7 size 103x20; Text 'Pezzi Al Minuto'
   IOField "campoIoNumeroAttvazioniAttuatori" at 197,329 size 96x32; FormatPattern s99999
      ProcessValue <- "0-DB-Generale_0-MinutiDiLavoro"
   TextField "campoTestoNumeroAttivazioniAttuatori" at 197,304 size 586x20; Text 'Numero Attivazioni Attuatori (legato a minuti di lavoro, tipo array di int non supportato?)'
   IOField "campoIoNumeroAttvazioniSensori" at 197,398 size 96x32; FormatPattern s99999
      ProcessValue <- "0-DB-Generale_0-MinutiDiLavoro"
   TextField "campoTestoNumeroAttivazioniSensori" at 197,373 size 573x20; Text 'Numero Attivazioni Sensori (legato a minuti di lavoro, tipo array di int non supportato?)'
*)